LIN {X -0.082,Y -167.901,Z 1787.358,A 0.000,B 0.000,C 90.000,E1 244.409} C_DIS
LIN {X 0.085,Y -166.640,Z 1787.348,A 0.000,B 0.000,C 90.000,E1 242.615} C_DIS
LIN {X -0.008,Y -162.626,Z 1787.324,A 0.000,B 0.000,C 90.000,E1 238.280} C_DIS
LIN {X 0.050,Y -161.313,Z 1787.314,A 0.000,B 0.000,C 90.000,E1 236.501} C_DIS
LIN {X -0.040,Y -157.310,Z 1787.289,A 0.000,B 0.000,C 90.000,E1 232.110} C_DIS
LIN {X -0.106,Y -155.287,Z 1787.275,A 0.000,B 0.000,C 90.000,E1 229.461} C_DIS
LIN {X 0.041,Y -151.650,Z 1787.250,A 0.000,B 0.000,C 90.000,E1 224.919} C_DIS
LIN {X -0.022,Y -150.518,Z 1787.240,A 0.000,B 0.000,C 90.000,E1 223.137} C_DIS
LIN {X 0.001,Y -147.243,Z 1787.214,A 0.000,B 0.000,C 90.000,E1 218.588} C_DIS
LIN {X -0.034,Y -145.267,Z 1787.194,A 0.000,B 0.000,C 90.000,E1 214.945} C_DIS
LIN {X 0.000,Y -142.375,Z 1787.163,A 0.000,B 0.000,C 90.000,E1 209.411} C_DIS
LIN {X 0.049,Y -141.351,Z 1787.148,A 0.000,B 0.000,C 90.000,E1 206.616} C_DIS
LIN {X 0.033,Y -139.340,Z 1787.112,A 0.000,B 0.000,C 90.000,E1 200.120} C_DIS
LIN {X 0.082,Y -139.006,Z 1787.101,A 0.000,B 0.000,C 90.000,E1 198.236} C_DIS
LIN {X 0.039,Y -138.339,Z 1787.055,A 0.000,B 0.000,C 90.000,E1 189.849} C_DIS
LIN {X 0.061,Y -139.404,Z 1787.008,A 0.000,B 0.000,C 90.000,E1 181.432} C_DIS
LIN {X -0.025,Y -141.312,Z 1786.972,A 0.000,B 0.000,C 90.000,E1 174.951} C_DIS
LIN {X -0.068,Y -142.671,Z 1786.956,A 0.000,B 0.000,C 90.000,E1 172.186} C_DIS
LIN {X 0.054,Y -145.021,Z 1786.931,A 0.000,B 0.000,C 90.000,E1 167.521} C_DIS
LIN {X 0.011,Y -147.648,Z 1786.910,A 0.000,B 0.000,C 90.000,E1 163.866} C_DIS
LIN {X -0.053,Y -150.283,Z 1786.890,A 0.000,B 0.000,C 90.000,E1 160.242} C_DIS
LIN {X -0.040,Y -153.688,Z 1786.870,A 0.000,B 0.000,C 90.000,E1 156.613} C_DIS
LIN {X 0.015,Y -157.102,Z 1786.850,A 0.000,B 0.000,C 90.000,E1 152.999} C_DIS
LIN {X -0.047,Y -161.242,Z 1786.830,A 0.000,B 0.000,C 90.000,E1 149.459} C_DIS
LIN {X 0.038,Y -163.329,Z 1786.820,A 0.000,B 0.000,C 90.000,E1 147.661} C_DIS
LIN {X -0.091,Y -167.782,Z 1786.801,A 0.000,B 0.000,C 90.000,E1 144.196} C_DIS
LIN {X 0.061,Y -171.597,Z 1786.786,A 0.000,B 0.000,C 90.000,E1 141.537} C_DIS
LIN {X -0.009,Y -176.549,Z 1786.767,A 0.000,B 0.000,C 90.000,E1 138.119} C_DIS
LIN {X -0.017,Y -180.848,Z 1786.753,A 0.000,B 0.000,C 90.000,E1 135.567} C_DIS
LIN {X -0.033,Y -186.259,Z 1786.734,A 0.000,B 0.000,C 90.000,E1 132.204} C_DIS
LIN {X -0.096,Y -190.895,Z 1786.721,A 0.000,B 0.000,C 90.000,E1 129.725} C_DIS
LIN {X 0.095,Y -196.660,Z 1786.702,A 0.000,B 0.000,C 90.000,E1 126.377} C_DIS
LIN {X 0.013,Y -199.902,Z 1786.693,A 0.000,B 0.000,C 90.000,E1 124.771} C_DIS
LIN {X 0.045,Y -204.295,Z 1786.680,A 0.000,B 0.000,C 90.000,E1 122.339} C_DIS
LIN {X 0.080,Y -210.742,Z 1786.662,A 0.000,B 0.000,C 90.000,E1 119.077} C_DIS
LIN {X 0.011,Y -211.127,Z 1786.660,A 0.000,B 0.000,C 90.000,E1 118.871} C_DIS
LIN {X -0.018,Y -337.494,Z 1786.660,A 0.000,B 0.000,C 90.000,E1 118.871} C_DIS
LIN {X 0.027,Y -340.375,Z 1786.660,A 0.000,B 0.000,C 90.000,E1 118.821} C_DIS
LIN {X -0.117,Y -345.110,Z 1786.659,A 0.000,B 0.000,C 90.000,E1 118.615} C_DIS
LIN {X 0.042,Y -347.762,Z 1786.658,A 0.000,B 0.000,C 90.000,E1 118.359} C_DIS
LIN {X -0.138,Y -351.455,Z 1786.655,A 0.000,B 0.000,C 90.000,E1 117.897} C_DIS
LIN {X 0.053,Y -354.388,Z 1786.651,A 0.000,B 0.000,C 90.000,E1 117.257} C_DIS
LIN {X 0.173,Y -369.809,Z 1786.633,A 0.000,B 0.000,C 90.000,E1 113.951} C_DIS
LIN {X -0.041,Y -383.135,Z 1786.619,A 0.000,B 0.000,C 90.000,E1 111.354} C_DIS
LIN {X -0.205,Y -395.265,Z 1786.606,A 0.000,B 0.000,C 90.000,E1 109.087} C_DIS
LIN {X -0.242,Y -404.241,Z 1786.596,A 0.000,B 0.000,C 90.000,E1 107.402} C_DIS
LIN {X -0.047,Y -409.915,Z 1786.590,A 0.000,B 0.000,C 90.000,E1 106.260} C_DIS
LIN {X -0.008,Y -413.783,Z 1786.586,A 0.000,B 0.000,C 90.000,E1 105.426} C_DIS
LIN {X 0.107,Y -414.948,Z 1786.584,A 0.000,B 0.000,C 90.000,E1 105.134} C_DIS
LIN {X 0.061,Y -416.955,Z 1786.581,A 0.000,B 0.000,C 90.000,E1 104.592} C_DIS
LIN {X -0.085,Y -418.203,Z 1786.578,A 0.000,B 0.000,C 90.000,E1 104.064} C_DIS
LIN {X -0.218,Y -417.913,Z 1786.575,A 0.000,B 0.000,C 90.000,E1 103.536} C_DIS
LIN {X -0.102,Y -414.004,Z 1786.536,A 0.000,B 0.000,C 90.000,E1 96.543} C_DIS
LIN {X -0.164,Y -414.009,Z 1786.536,A 0.000,B 0.000,C 90.000,E1 96.543} C_DIS
LIN {X -0.056,Y -438.067,Z 1786.526,A 0.000,B 0.000,C 90.000,E1 94.702} C_DIS
LIN {X -0.081,Y -442.270,Z 1786.524,A 0.000,B 0.000,C 90.000,E1 94.302} C_DIS
LIN {X -0.189,Y -443.992,Z 1786.522,A 0.000,B 0.000,C 90.000,E1 94.069} C_DIS
LIN {X 0.112,Y -445.315,Z 1786.521,A 0.000,B 0.000,C 90.000,E1 93.784} C_DIS
LIN {X 0.030,Y -447.152,Z 1786.518,A 0.000,B 0.000,C 90.000,E1 93.269} C_DIS
LIN {X -0.018,Y -447.927,Z 1786.515,A 0.000,B 0.000,C 90.000,E1 92.751} C_DIS
LIN {X -0.078,Y -447.768,Z 1786.512,A 0.000,B 0.000,C 90.000,E1 92.236} C_DIS
LIN {X -0.117,Y -446.654,Z 1786.510,A 0.000,B 0.000,C 90.000,E1 91.718} C_DIS
LIN {X 0.078,Y -445.692,Z 1786.508,A 0.000,B 0.000,C 90.000,E1 91.432} C_DIS
LIN {X -0.171,Y -444.401,Z 1786.507,A 0.000,B 0.000,C 90.000,E1 91.203} C_DIS
LIN {X 0.183,Y -432.865,Z 1786.496,A 0.000,B 0.000,C 90.000,E1 89.312} C_DIS
LIN {X 0.182,Y -422.902,Z 1786.487,A 0.000,B 0.000,C 90.000,E1 87.707} C_DIS
LIN {X -0.204,Y -419.006,Z 1786.484,A 0.000,B 0.000,C 90.000,E1 87.135} C_DIS
LIN {X 0.152,Y -419.014,Z 1786.484,A 0.000,B 0.000,C 90.000,E1 87.078} C_DIS
LIN {X -0.079,Y -421.363,Z 1786.474,A 0.000,B 0.000,C 90.000,E1 85.298} C_DIS
LIN {X 0.158,Y -421.920,Z 1786.471,A 0.000,B 0.000,C 90.000,E1 84.723} C_DIS
LIN {X -0.020,Y -421.140,Z 1786.468,A 0.000,B 0.000,C 90.000,E1 84.204} C_DIS
LIN {X -0.192,Y -419.699,Z 1786.465,A 0.000,B 0.000,C 90.000,E1 83.685} C_DIS
LIN {X 0.047,Y -417.913,Z 1786.462,A 0.000,B 0.000,C 90.000,E1 83.109} C_DIS
LIN {X 0.133,Y -413.778,Z 1786.456,A 0.000,B 0.000,C 90.000,E1 82.008} C_DIS
LIN {X -0.185,Y -408.002,Z 1786.448,A 0.000,B 0.000,C 90.000,E1 80.679} C_DIS
LIN {X 0.058,Y -399.400,Z 1786.437,A 0.000,B 0.000,C 90.000,E1 78.701} C_DIS
LIN {X -0.110,Y -390.545,Z 1786.426,A 0.000,B 0.000,C 90.000,E1 76.756} C_DIS
LIN {X -0.075,Y -381.580,Z 1786.415,A 0.000,B 0.000,C 90.000,E1 74.755} C_DIS
LIN {X -0.040,Y -372.591,Z 1786.404,A 0.000,B 0.000,C 90.000,E1 72.725} C_DIS
LIN {X -0.081,Y -363.547,Z 1786.393,A 0.000,B 0.000,C 90.000,E1 70.678} C_DIS
LIN {X -0.076,Y -354.371,Z 1786.381,A 0.000,B 0.000,C 90.000,E1 68.592} C_DIS
LIN {X -0.155,Y -346.485,Z 1786.371,A 0.000,B 0.000,C 90.000,E1 66.794} C_DIS
LIN {X -0.098,Y -335.869,Z 1786.357,A 0.000,B 0.000,C 90.000,E1 64.332} C_DIS
LIN {X 0.061,Y -327.934,Z 1786.347,A 0.000,B 0.000,C 90.000,E1 62.436} C_DIS
LIN {X 0.073,Y -319.703,Z 1786.336,A 0.000,B 0.000,C 90.000,E1 60.539} C_DIS
LIN {X 0.090,Y -311.024,Z 1786.326,A 0.000,B 0.000,C 90.000,E1 58.614} C_DIS
LIN {X -0.149,Y -302.097,Z 1786.315,A 0.000,B 0.000,C 90.000,E1 56.707} C_DIS
LIN {X 0.034,Y -291.535,Z 1786.302,A 0.000,B 0.000,C 90.000,E1 54.356} C_DIS
LIN {X 0.051,Y -277.134,Z 1786.283,A 0.000,B 0.000,C 90.000,E1 50.964} C_DIS
LIN {X 0.048,Y -265.046,Z 1786.266,A 0.000,B 0.000,C 90.000,E1 47.838} C_DIS
LIN {X 0.015,Y -256.155,Z 1786.252,A 0.000,B 0.000,C 90.000,E1 45.364} C_DIS
LIN {X -0.042,Y -245.127,Z 1786.234,A 0.000,B 0.000,C 90.000,E1 42.123} C_DIS
LIN {X 0.016,Y -234.692,Z 1786.215,A 0.000,B 0.000,C 90.000,E1 38.785} C_DIS
LIN {X -0.115,Y -225.884,Z 1786.199,A 0.000,B 0.000,C 90.000,E1 35.804} C_DIS
LIN {X 0.031,Y -217.527,Z 1786.182,A 0.000,B 0.000,C 90.000,E1 32.704} C_DIS
LIN {X 0.027,Y -209.871,Z 1786.164,A 0.000,B 0.000,C 90.000,E1 29.589} C_DIS
LIN {X -0.029,Y -202.778,Z 1786.147,A 0.000,B 0.000,C 90.000,E1 26.437} C_DIS
LIN {X 0.022,Y -196.511,Z 1786.129,A 0.000,B 0.000,C 90.000,E1 23.206} C_DIS
LIN {X 0.044,Y -191.090,Z 1786.111,A 0.000,B 0.000,C 90.000,E1 19.939} C_DIS
LIN {X -0.077,Y -186.595,Z 1786.093,A 0.000,B 0.000,C 90.000,E1 16.677} C_DIS
LIN {X 0.071,Y -183.018,Z 1786.074,A 0.000,B 0.000,C 90.000,E1 13.300} C_DIS
LIN {X -0.098,Y -179.575,Z 1786.051,A 0.000,B 0.000,C 90.000,E1 9.151} C_DIS
LIN {X 0.079,Y -176.772,Z 1786.022,A 0.000,B 0.000,C 90.000,E1 4.012} C_DIS
LIN {X 0.045,Y -175.198,Z 1785.978,A 0.000,B 0.000,C 90.000,E1 356.102} C_DIS
LIN {X -0.039,Y -175.639,Z 1785.945,A 0.000,B 0.000,C 90.000,E1 350.151} C_DIS
LIN {X -0.007,Y -177.753,Z 1785.907,A 0.000,B 0.000,C 90.000,E1 343.323} C_DIS
LIN {X 0.010,Y -180.661,Z 1785.879,A 0.000,B 0.000,C 90.000,E1 338.230} C_DIS
LIN {X 0.016,Y -184.417,Z 1785.851,A 0.000,B 0.000,C 90.000,E1 333.179} C_DIS
LIN {X 0.042,Y -188.378,Z 1785.828,A 0.000,B 0.000,C 90.000,E1 328.997} C_DIS
LIN {X -0.070,Y -193.294,Z 1785.805,A 0.000,B 0.000,C 90.000,E1 324.895} C_DIS
LIN {X -0.058,Y -198.263,Z 1785.787,A 0.000,B 0.000,C 90.000,E1 321.618} C_DIS
LIN {X -0.021,Y -202.721,Z 1785.773,A 0.000,B 0.000,C 90.000,E1 319.175} C_DIS
LIN {X -0.077,Y -207.911,Z 1785.760,A 0.000,B 0.000,C 90.000,E1 316.782} C_DIS
LIN {X 0.113,Y -213.920,Z 1785.747,A 0.000,B 0.000,C 90.000,E1 314.352} C_DIS
LIN {X -0.080,Y -219.742,Z 1785.736,A 0.000,B 0.000,C 90.000,E1 312.447} C_DIS
LIN {X 0.064,Y -225.118,Z 1785.727,A 0.000,B 0.000,C 90.000,E1 310.862} C_DIS
LIN {X -0.093,Y -232.803,Z 1785.716,A 0.000,B 0.000,C 90.000,E1 308.991} C_DIS
LIN {X 0.081,Y -239.780,Z 1785.708,A 0.000,B 0.000,C 90.000,E1 307.443} C_DIS
LIN {X 0.052,Y -251.469,Z 1785.696,A 0.000,B 0.000,C 90.000,E1 305.231} C_DIS
LIN {X -0.046,Y -264.356,Z 1785.684,A 0.000,B 0.000,C 90.000,E1 303.086} C_DIS
LIN {X 0.077,Y -283.080,Z 1785.668,A 0.000,B 0.000,C 90.000,E1 300.256} C_DIS
LIN {X 0.015,Y -300.593,Z 1785.655,A 0.000,B 0.000,C 90.000,E1 297.897} C_DIS
LIN {X 0.114,Y -318.945,Z 1785.642,A 0.000,B 0.000,C 90.000,E1 295.591} C_DIS
LIN {X -0.054,Y -332.172,Z 1785.633,A 0.000,B 0.000,C 90.000,E1 294.027} C_DIS
LIN {X -0.015,Y -344.484,Z 1785.625,A 0.000,B 0.000,C 90.000,E1 292.514} C_DIS
LIN {X 0.041,Y -354.474,Z 1785.618,A 0.000,B 0.000,C 90.000,E1 291.280} C_DIS
LIN {X 0.098,Y -363.916,Z 1785.612,A 0.000,B 0.000,C 90.000,E1 290.066} C_DIS
LIN {X -0.153,Y -370.378,Z 1785.607,A 0.000,B 0.000,C 90.000,E1 289.214} C_DIS
LIN {X -0.001,Y -376.050,Z 1785.602,A 0.000,B 0.000,C 90.000,E1 288.308} C_DIS
LIN {X 0.213,Y -379.294,Z 1785.599,A 0.000,B 0.000,C 90.000,E1 287.692} C_DIS
LIN {X -0.033,Y -382.098,Z 1785.595,A 0.000,B 0.000,C 90.000,E1 287.149} C_DIS
LIN {X -0.007,Y -384.499,Z 1785.592,A 0.000,B 0.000,C 90.000,E1 286.567} C_DIS
LIN {X 0.150,Y -386.517,Z 1785.589,A 0.000,B 0.000,C 90.000,E1 285.969} C_DIS
LIN {X -0.061,Y -388.166,Z 1785.586,A 0.000,B 0.000,C 90.000,E1 285.426} C_DIS
LIN {X 0.113,Y -389.485,Z 1785.583,A 0.000,B 0.000,C 90.000,E1 284.828} C_DIS
LIN {X -0.180,Y -390.422,Z 1785.579,A 0.000,B 0.000,C 90.000,E1 284.300} C_DIS
LIN {X 0.008,Y -391.016,Z 1785.576,A 0.000,B 0.000,C 90.000,E1 283.703} C_DIS
LIN {X 0.110,Y -391.223,Z 1785.573,A 0.000,B 0.000,C 90.000,E1 283.119} C_DIS
LIN {X -0.164,Y -391.064,Z 1785.570,A 0.000,B 0.000,C 90.000,E1 282.591} C_DIS
LIN {X -0.054,Y -390.576,Z 1785.567,A 0.000,B 0.000,C 90.000,E1 282.007} C_DIS
LIN {X 0.056,Y -389.758,Z 1785.563,A 0.000,B 0.000,C 90.000,E1 281.422} C_DIS
LIN {X 0.162,Y -388.564,Z 1785.560,A 0.000,B 0.000,C 90.000,E1 280.838} C_DIS
LIN {X -0.120,Y -387.029,Z 1785.557,A 0.000,B 0.000,C 90.000,E1 280.310} C_DIS
LIN {X -0.052,Y -384.062,Z 1785.552,A 0.000,B 0.000,C 90.000,E1 279.443} C_DIS
LIN {X 0.051,Y -380.355,Z 1785.548,A 0.000,B 0.000,C 90.000,E1 278.568} C_DIS
LIN {X 0.055,Y -375.850,Z 1785.543,A 0.000,B 0.000,C 90.000,E1 277.701} C_DIS
LIN {X 0.024,Y -370.428,Z 1785.538,A 0.000,B 0.000,C 90.000,E1 276.834} C_DIS
LIN {X -0.037,Y -366.343,Z 1785.535,A 0.000,B 0.000,C 90.000,E1 276.258} C_DIS
LIN {X -0.119,Y -361.714,Z 1785.531,A 0.000,B 0.000,C 90.000,E1 275.682} C_DIS
LIN {X 0.129,Y -356.504,Z 1785.528,A 0.000,B 0.000,C 90.000,E1 275.049} C_DIS
LIN {X 0.065,Y -350.776,Z 1785.525,A 0.000,B 0.000,C 90.000,E1 274.473} C_DIS
LIN {X 0.104,Y -341.958,Z 1785.521,A 0.000,B 0.000,C 90.000,E1 273.669} C_DIS
LIN {X -0.056,Y -335.894,Z 1785.518,A 0.000,B 0.000,C 90.000,E1 273.212} C_DIS
LIN {X -0.008,Y -329.703,Z 1785.515,A 0.000,B 0.000,C 90.000,E1 272.751} C_DIS
LIN {X -0.105,Y -323.138,Z 1785.513,A 0.000,B 0.000,C 90.000,E1 272.350} C_DIS
LIN {X 0.043,Y -316.460,Z 1785.511,A 0.000,B 0.000,C 90.000,E1 271.949} C_DIS
LIN {X 0.136,Y -309.448,Z 1785.509,A 0.000,B 0.000,C 90.000,E1 271.604} C_DIS
LIN {X -0.089,Y -301.903,Z 1785.508,A 0.000,B 0.000,C 90.000,E1 271.375} C_DIS
LIN {X -0.015,Y -294.587,Z 1785.506,A 0.000,B 0.000,C 90.000,E1 271.146} C_DIS
LIN {X 0.115,Y -283.709,Z 1785.505,A 0.000,B 0.000,C 90.000,E1 270.859} C_DIS
LIN {X 0.130,Y -268.696,Z 1785.503,A 0.000,B 0.000,C 90.000,E1 270.573} C_DIS
LIN {X 0.081,Y -256.288,Z 1785.502,A 0.000,B 0.000,C 90.000,E1 270.401} C_DIS
LIN {X -0.121,Y -245.286,Z 1785.502,A 0.000,B 0.000,C 90.000,E1 270.344} C_DIS
LIN {X -0.078,Y -229.736,Z 1785.501,A 0.000,B 0.000,C 90.000,E1 270.286} C_DIS
LIN {X -0.083,Y -181.581,Z 1785.501,A 0.000,B 0.000,C 90.000,E1 270.286} C_DIS
LIN {X 0.088,Y -180.826,Z 1785.471,A 0.000,B 0.000,C 90.000,E1 264.837} C_DIS
LIN {X -0.012,Y -178.930,Z 1785.443,A 0.000,B 0.000,C 90.000,E1 259.803} C_DIS
LIN {X 0.026,Y -175.979,Z 1785.415,A 0.000,B 0.000,C 90.000,E1 254.700} C_DIS
LIN {X -0.028,Y -175.469,Z 1785.410,A 0.000,B 0.000,C 90.000,E1 253.866} C_DIS
LIN {X 0.028,Y -172.218,Z 1785.387,A 0.000,B 0.000,C 90.000,E1 249.571} C_DIS
LIN {X 0.006,Y -171.693,Z 1785.382,A 0.000,B 0.000,C 90.000,E1 248.720} C_DIS
LIN {X 0.081,Y -167.288,Z 1785.353,A 0.000,B 0.000,C 90.000,E1 243.512} C_DIS
LIN {X 0.014,Y -166.664,Z 1785.348,A 0.000,B 0.000,C 90.000,E1 242.666} C_DIS
LIN {X -0.070,Y -162.647,Z 1785.324,A 0.000,B 0.000,C 90.000,E1 238.329} C_DIS
LIN {X -0.008,Y -161.335,Z 1785.314,A 0.000,B 0.000,C 90.000,E1 236.548} C_DIS
LIN {X 0.035,Y -157.331,Z 1785.290,A 0.000,B 0.000,C 90.000,E1 232.110} C_DIS
LIN {X -0.032,Y -155.313,Z 1785.275,A 0.000,B 0.000,C 90.000,E1 229.461} C_DIS
LIN {X 0.007,Y -151.669,Z 1785.250,A 0.000,B 0.000,C 90.000,E1 224.960} C_DIS
LIN {X -0.053,Y -150.534,Z 1785.240,A 0.000,B 0.000,C 90.000,E1 223.176} C_DIS
LIN {X -0.020,Y -147.259,Z 1785.214,A 0.000,B 0.000,C 90.000,E1 218.624} C_DIS
LIN {X 0.037,Y -145.286,Z 1785.194,A 0.000,B 0.000,C 90.000,E1 214.945} C_DIS
LIN {X 0.071,Y -142.386,Z 1785.164,A 0.000,B 0.000,C 90.000,E1 209.411} C_DIS
LIN {X -0.007,Y -141.364,Z 1785.148,A 0.000,B 0.000,C 90.000,E1 206.668} C_DIS
LIN {X -0.028,Y -139.344,Z 1785.112,A 0.000,B 0.000,C 90.000,E1 200.174} C_DIS
LIN {X -0.023,Y -139.014,Z 1785.102,A 0.000,B 0.000,C 90.000,E1 198.308} C_DIS
LIN {X -0.028,Y -138.341,Z 1785.055,A 0.000,B 0.000,C 90.000,E1 189.905} C_DIS
LIN {X -0.008,Y -139.397,Z 1785.008,A 0.000,B 0.000,C 90.000,E1 181.489} C_DIS
LIN {X 0.045,Y -141.298,Z 1784.972,A 0.000,B 0.000,C 90.000,E1 174.951} C_DIS
LIN {X 0.003,Y -142.660,Z 1784.957,A 0.000,B 0.000,C 90.000,E1 172.186} C_DIS
LIN {X -0.047,Y -145.004,Z 1784.931,A 0.000,B 0.000,C 90.000,E1 167.589} C_DIS
LIN {X -0.057,Y -147.631,Z 1784.911,A 0.000,B 0.000,C 90.000,E1 163.921} C_DIS
LIN {X 0.020,Y -150.260,Z 1784.890,A 0.000,B 0.000,C 90.000,E1 160.242} C_DIS
LIN {X 0.033,Y -153.659,Z 1784.870,A 0.000,B 0.000,C 90.000,E1 156.613} C_DIS
LIN {X -0.050,Y -157.074,Z 1784.850,A 0.000,B 0.000,C 90.000,E1 153.050} C_DIS
LIN {X 0.029,Y -161.207,Z 1784.830,A 0.000,B 0.000,C 90.000,E1 149.459} C_DIS
LIN {X -0.023,Y -163.298,Z 1784.821,A 0.000,B 0.000,C 90.000,E1 147.709} C_DIS
LIN {X -0.013,Y -167.745,Z 1784.801,A 0.000,B 0.000,C 90.000,E1 144.196} C_DIS
LIN {X -0.101,Y -171.562,Z 1784.787,A 0.000,B 0.000,C 90.000,E1 141.618} C_DIS
LIN {X -0.060,Y -176.508,Z 1784.767,A 0.000,B 0.000,C 90.000,E1 138.162} C_DIS
LIN {X 0.065,Y -180.806,Z 1784.753,A 0.000,B 0.000,C 90.000,E1 135.567} C_DIS
LIN {X 0.051,Y -186.214,Z 1784.734,A 0.000,B 0.000,C 90.000,E1 132.204} C_DIS
LIN {X -0.011,Y -190.851,Z 1784.721,A 0.000,B 0.000,C 90.000,E1 129.725} C_DIS
LIN {X 0.023,Y -196.612,Z 1784.702,A 0.000,B 0.000,C 90.000,E1 126.423} C_DIS
LIN {X -0.064,Y -199.850,Z 1784.693,A 0.000,B 0.000,C 90.000,E1 124.818} C_DIS
LIN {X 0.132,Y -204.249,Z 1784.680,A 0.000,B 0.000,C 90.000,E1 122.339} C_DIS
LIN {X -0.043,Y -210.799,Z 1784.661,A 0.000,B 0.000,C 90.000,E1 119.077} C_DIS
LIN {X -0.001,Y -211.085,Z 1784.661,A 0.000,B 0.000,C 90.000,E1 118.899} C_DIS
LIN {X 0.125,Y -337.558,Z 1784.661,A 0.000,B 0.000,C 90.000,E1 118.871} C_DIS
LIN {X -0.126,Y -340.364,Z 1784.660,A 0.000,B 0.000,C 90.000,E1 118.871} C_DIS
LIN {X 0.030,Y -345.120,Z 1784.659,A 0.000,B 0.000,C 90.000,E1 118.615} C_DIS
LIN {X 0.189,Y -347.789,Z 1784.658,A 0.000,B 0.000,C 90.000,E1 118.359} C_DIS
LIN {X 0.024,Y -351.493,Z 1784.655,A 0.000,B 0.000,C 90.000,E1 117.897} C_DIS
LIN {X -0.097,Y -354.485,Z 1784.652,A 0.000,B 0.000,C 90.000,E1 117.308} C_DIS
LIN {X 0.015,Y -370.423,Z 1784.633,A 0.000,B 0.000,C 90.000,E1 114.003} C_DIS
LIN {X -0.053,Y -385.844,Z 1784.617,A 0.000,B 0.000,C 90.000,E1 111.099} C_DIS
LIN {X 0.221,Y -398.629,Z 1784.604,A 0.000,B 0.000,C 90.000,E1 108.779} C_DIS
LIN {X -0.048,Y -409.855,Z 1784.594,A 0.000,B 0.000,C 90.000,E1 106.858} C_DIS
LIN {X -0.059,Y -417.583,Z 1784.586,A 0.000,B 0.000,C 90.000,E1 105.481} C_DIS
LIN {X 0.189,Y -423.245,Z 1784.580,A 0.000,B 0.000,C 90.000,E1 104.356} C_DIS
LIN {X -0.174,Y -426.788,Z 1784.575,A 0.000,B 0.000,C 90.000,E1 103.592} C_DIS
LIN {X 0.159,Y -428.400,Z 1784.572,A 0.000,B 0.000,C 90.000,E1 103.008} C_DIS
LIN {X 0.084,Y -428.529,Z 1784.569,A 0.000,B 0.000,C 90.000,E1 102.479} C_DIS
LIN {X -0.001,Y -425.481,Z 1784.531,A 0.000,B 0.000,C 90.000,E1 95.625} C_DIS
LIN {X -0.063,Y -425.532,Z 1784.531,A 0.000,B 0.000,C 90.000,E1 95.625} C_DIS
LIN {X 0.160,Y -438.457,Z 1784.526,A 0.000,B 0.000,C 90.000,E1 94.645} C_DIS
LIN {X 0.132,Y -442.495,Z 1784.524,A 0.000,B 0.000,C 90.000,E1 94.245} C_DIS
LIN {X -0.029,Y -444.200,Z 1784.522,A 0.000,B 0.000,C 90.000,E1 94.012} C_DIS
LIN {X 0.222,Y -445.501,Z 1784.521,A 0.000,B 0.000,C 90.000,E1 93.726} C_DIS
LIN {X 0.143,Y -447.240,Z 1784.518,A 0.000,B 0.000,C 90.000,E1 93.212} C_DIS
LIN {X 0.095,Y -447.934,Z 1784.515,A 0.000,B 0.000,C 90.000,E1 92.694} C_DIS
LIN {X 0.037,Y -447.698,Z 1784.512,A 0.000,B 0.000,C 90.000,E1 92.178} C_DIS
LIN {X -0.003,Y -446.501,Z 1784.509,A 0.000,B 0.000,C 90.000,E1 91.661} C_DIS
LIN {X 0.192,Y -445.487,Z 1784.508,A 0.000,B 0.000,C 90.000,E1 91.375} C_DIS
LIN {X -0.058,Y -444.135,Z 1784.506,A 0.000,B 0.000,C 90.000,E1 91.146} C_DIS
LIN {X 0.012,Y -430.944,Z 1784.495,A 0.000,B 0.000,C 90.000,E1 89.026} C_DIS
LIN {X 0.149,Y -428.919,Z 1784.493,A 0.000,B 0.000,C 90.000,E1 88.682} C_DIS
LIN {X 0.086,Y -428.916,Z 1784.493,A 0.000,B 0.000,C 90.000,E1 88.682} C_DIS
LIN {X 0.132,Y -431.582,Z 1784.480,A 0.000,B 0.000,C 90.000,E1 86.331} C_DIS
LIN {X 0.006,Y -431.150,Z 1784.477,A 0.000,B 0.000,C 90.000,E1 85.812} C_DIS
LIN {X -0.149,Y -429.813,Z 1784.474,A 0.000,B 0.000,C 90.000,E1 85.298} C_DIS
LIN {X 0.154,Y -428.077,Z 1784.471,A 0.000,B 0.000,C 90.000,E1 84.723} C_DIS
LIN {X -0.113,Y -423.922,Z 1784.465,A 0.000,B 0.000,C 90.000,E1 83.685} C_DIS
LIN {X 0.131,Y -418.011,Z 1784.457,A 0.000,B 0.000,C 90.000,E1 82.299} C_DIS
LIN {X -0.010,Y -410.399,Z 1784.448,A 0.000,B 0.000,C 90.000,E1 80.679} C_DIS
LIN {X -0.116,Y -401.212,Z 1784.438,A 0.000,B 0.000,C 90.000,E1 78.757} C_DIS
LIN {X 0.138,Y -391.925,Z 1784.427,A 0.000,B 0.000,C 90.000,E1 76.756} C_DIS
LIN {X -0.175,Y -382.606,Z 1784.416,A 0.000,B 0.000,C 90.000,E1 74.810} C_DIS
LIN {X -0.113,Y -373.295,Z 1784.404,A 0.000,B 0.000,C 90.000,E1 72.779} C_DIS
LIN {X -0.136,Y -363.958,Z 1784.393,A 0.000,B 0.000,C 90.000,E1 70.732} C_DIS
LIN {X -0.118,Y -354.476,Z 1784.381,A 0.000,B 0.000,C 90.000,E1 68.646} C_DIS
LIN {X 0.155,Y -344.991,Z 1784.370,A 0.000,B 0.000,C 90.000,E1 66.485} C_DIS
LIN {X 0.163,Y -334.332,Z 1784.356,A 0.000,B 0.000,C 90.000,E1 64.024} C_DIS
LIN {X 0.096,Y -325.026,Z 1784.344,A 0.000,B 0.000,C 90.000,E1 61.847} C_DIS
LIN {X 0.133,Y -318.110,Z 1784.335,A 0.000,B 0.000,C 90.000,E1 60.255} C_DIS
LIN {X 0.125,Y -309.395,Z 1784.324,A 0.000,B 0.000,C 90.000,E1 58.329} C_DIS
LIN {X -0.139,Y -300.441,Z 1784.313,A 0.000,B 0.000,C 90.000,E1 56.421} C_DIS
LIN {X 0.161,Y -288.413,Z 1784.299,A 0.000,B 0.000,C 90.000,E1 53.703} C_DIS
LIN {X -0.026,Y -275.631,Z 1784.281,A 0.000,B 0.000,C 90.000,E1 50.678} C_DIS
LIN {X -0.067,Y -263.620,Z 1784.264,A 0.000,B 0.000,C 90.000,E1 47.553} C_DIS
LIN {X -0.138,Y -254.720,Z 1784.250,A 0.000,B 0.000,C 90.000,E1 45.081} C_DIS
LIN {X 0.129,Y -243.722,Z 1784.232,A 0.000,B 0.000,C 90.000,E1 41.757} C_DIS
LIN {X -0.041,Y -233.331,Z 1784.214,A 0.000,B 0.000,C 90.000,E1 38.463} C_DIS
LIN {X 0.100,Y -223.514,Z 1784.195,A 0.000,B 0.000,C 90.000,E1 35.025} C_DIS
LIN {X -0.122,Y -215.301,Z 1784.178,A 0.000,B 0.000,C 90.000,E1 32.005} C_DIS
LIN {X 0.076,Y -207.787,Z 1784.160,A 0.000,B 0.000,C 90.000,E1 28.821} C_DIS
LIN {X -0.027,Y -200.844,Z 1784.143,A 0.000,B 0.000,C 90.000,E1 25.668} C_DIS
LIN {X -0.104,Y -194.784,Z 1784.125,A 0.000,B 0.000,C 90.000,E1 22.461} C_DIS
LIN {X 0.055,Y -189.569,Z 1784.106,A 0.000,B 0.000,C 90.000,E1 19.141} C_DIS
LIN {X 0.017,Y -185.305,Z 1784.088,A 0.000,B 0.000,C 90.000,E1 15.843} C_DIS
LIN {X -0.090,Y -181.927,Z 1784.069,A 0.000,B 0.000,C 90.000,E1 12.535} C_DIS
LIN {X -0.052,Y -178.155,Z 1784.041,A 0.000,B 0.000,C 90.000,E1 7.466} C_DIS
LIN {X 0.029,Y -175.619,Z 1784.008,A 0.000,B 0.000,C 90.000,E1 1.489} C_DIS
LIN {X -0.083,Y -174.896,Z 1783.969,A 0.000,B 0.000,C 90.000,E1 354.432} C_DIS
LIN {X 0.043,Y -175.660,Z 1783.936,A 0.000,B 0.000,C 90.000,E1 348.409} C_DIS
LIN {X -0.041,Y -177.863,Z 1783.903,A 0.000,B 0.000,C 90.000,E1 342.472} C_DIS
LIN {X 0.049,Y -180.967,Z 1783.874,A 0.000,B 0.000,C 90.000,E1 337.358} C_DIS
LIN {X -0.102,Y -184.893,Z 1783.846,A 0.000,B 0.000,C 90.000,E1 332.359} C_DIS
LIN {X 0.020,Y -189.093,Z 1783.823,A 0.000,B 0.000,C 90.000,E1 328.152} C_DIS
LIN {X 0.014,Y -193.188,Z 1783.805,A 0.000,B 0.000,C 90.000,E1 324.848} C_DIS
LIN {X -0.014,Y -198.208,Z 1783.786,A 0.000,B 0.000,C 90.000,E1 321.582} C_DIS
LIN {X 0.030,Y -202.742,Z 1783.773,A 0.000,B 0.000,C 90.000,E1 319.138} C_DIS
LIN {X -0.018,Y -207.992,Z 1783.760,A 0.000,B 0.000,C 90.000,E1 316.743} C_DIS
LIN {X 0.029,Y -214.066,Z 1783.746,A 0.000,B 0.000,C 90.000,E1 314.352} C_DIS
LIN {X -0.002,Y -219.915,Z 1783.736,A 0.000,B 0.000,C 90.000,E1 312.405} C_DIS
LIN {X -0.020,Y -225.319,Z 1783.727,A 0.000,B 0.000,C 90.000,E1 310.862} C_DIS
LIN {X 0.025,Y -231.402,Z 1783.719,A 0.000,B 0.000,C 90.000,E1 309.322} C_DIS
LIN {X 0.031,Y -238.200,Z 1783.710,A 0.000,B 0.000,C 90.000,E1 307.810} C_DIS
LIN {X -0.027,Y -249.701,Z 1783.698,A 0.000,B 0.000,C 90.000,E1 305.598} C_DIS
LIN {X -0.014,Y -262.453,Z 1783.686,A 0.000,B 0.000,C 90.000,E1 303.420} C_DIS
LIN {X 0.057,Y -281.001,Z 1783.670,A 0.000,B 0.000,C 90.000,E1 300.590} C_DIS
LIN {X -0.060,Y -298.477,Z 1783.657,A 0.000,B 0.000,C 90.000,E1 298.231} C_DIS
LIN {X 0.023,Y -319.431,Z 1783.642,A 0.000,B 0.000,C 90.000,E1 295.591} C_DIS
LIN {X 0.014,Y -332.627,Z 1783.633,A 0.000,B 0.000,C 90.000,E1 294.003} C_DIS
LIN {X -0.093,Y -345.424,Z 1783.625,A 0.000,B 0.000,C 90.000,E1 292.461} C_DIS
LIN {X -0.026,Y -355.423,Z 1783.618,A 0.000,B 0.000,C 90.000,E1 291.227} C_DIS
LIN {X 0.168,Y -364.840,Z 1783.611,A 0.000,B 0.000,C 90.000,E1 289.993} C_DIS
LIN {X -0.076,Y -371.240,Z 1783.606,A 0.000,B 0.000,C 90.000,E1 289.141} C_DIS
LIN {X -0.016,Y -375.093,Z 1783.603,A 0.000,B 0.000,C 90.000,E1 288.544} C_DIS
LIN {X 0.074,Y -378.476,Z 1783.600,A 0.000,B 0.000,C 90.000,E1 287.946} C_DIS
LIN {X -0.057,Y -382.770,Z 1783.595,A 0.000,B 0.000,C 90.000,E1 287.094} C_DIS
LIN {X 0.085,Y -385.132,Z 1783.592,A 0.000,B 0.000,C 90.000,E1 286.496} C_DIS
LIN {X -0.129,Y -387.094,Z 1783.589,A 0.000,B 0.000,C 90.000,E1 285.953} C_DIS
LIN {X -0.069,Y -388.730,Z 1783.585,A 0.000,B 0.000,C 90.000,E1 285.371} C_DIS
LIN {X 0.109,Y -390.012,Z 1783.582,A 0.000,B 0.000,C 90.000,E1 284.773} C_DIS
LIN {X -0.179,Y -390.889,Z 1783.579,A 0.000,B 0.000,C 90.000,E1 284.245} C_DIS
LIN {X 0.014,Y -391.436,Z 1783.576,A 0.000,B 0.000,C 90.000,E1 283.647} C_DIS
LIN {X 0.119,Y -391.600,Z 1783.573,A 0.000,B 0.000,C 90.000,E1 283.063} C_DIS
LIN {X -0.152,Y -391.417,Z 1783.569,A 0.000,B 0.000,C 90.000,E1 282.535} C_DIS
LIN {X -0.039,Y -390.884,Z 1783.566,A 0.000,B 0.000,C 90.000,E1 281.951} C_DIS
LIN {X 0.073,Y -390.019,Z 1783.563,A 0.000,B 0.000,C 90.000,E1 281.366} C_DIS
LIN {X -0.200,Y -388.800,Z 1783.560,A 0.000,B 0.000,C 90.000,E1 280.838} C_DIS
LIN {X -0.097,Y -387.221,Z 1783.557,A 0.000,B 0.000,C 90.000,E1 280.254} C_DIS
LIN {X 0.037,Y -384.206,Z 1783.552,A 0.000,B 0.000,C 90.000,E1 279.378} C_DIS
LIN {X 0.079,Y -380.399,Z 1783.547,A 0.000,B 0.000,C 90.000,E1 278.511} C_DIS
LIN {X 0.083,Y -375.819,Z 1783.542,A 0.000,B 0.000,C 90.000,E1 277.644} C_DIS
LIN {X 0.053,Y -370.357,Z 1783.538,A 0.000,B 0.000,C 90.000,E1 276.777} C_DIS
LIN {X -0.032,Y -363.938,Z 1783.533,A 0.000,B 0.000,C 90.000,E1 275.910} C_DIS
LIN {X 0.156,Y -356.263,Z 1783.528,A 0.000,B 0.000,C 90.000,E1 274.992} C_DIS
LIN {X 0.136,Y -350.544,Z 1783.525,A 0.000,B 0.000,C 90.000,E1 274.416} C_DIS
LIN {X -0.028,Y -344.525,Z 1783.522,A 0.000,B 0.000,C 90.000,E1 273.898} C_DIS
LIN {X 0.063,Y -338.495,Z 1783.519,A 0.000,B 0.000,C 90.000,E1 273.383} C_DIS
LIN {X 0.025,Y -332.294,Z 1783.516,A 0.000,B 0.000,C 90.000,E1 272.922} C_DIS
LIN {X 0.135,Y -325.776,Z 1783.514,A 0.000,B 0.000,C 90.000,E1 272.465} C_DIS
LIN {X -0.138,Y -319.039,Z 1783.512,A 0.000,B 0.000,C 90.000,E1 272.121} C_DIS
LIN {X -0.135,Y -312.082,Z 1783.510,A 0.000,B 0.000,C 90.000,E1 271.776} C_DIS
LIN {X 0.137,Y -304.768,Z 1783.508,A 0.000,B 0.000,C 90.000,E1 271.432} C_DIS
LIN {X 0.122,Y -297.423,Z 1783.507,A 0.000,B 0.000,C 90.000,E1 271.203} C_DIS
LIN {X -0.106,Y -286.602,Z 1783.505,A 0.000,B 0.000,C 90.000,E1 270.974} C_DIS
LIN {X -0.105,Y -275.330,Z 1783.504,A 0.000,B 0.000,C 90.000,E1 270.745} C_DIS
LIN {X 0.058,Y -263.582,Z 1783.503,A 0.000,B 0.000,C 90.000,E1 270.516} C_DIS
LIN {X 0.030,Y -254.121,Z 1783.502,A 0.000,B 0.000,C 90.000,E1 270.401} C_DIS
LIN {X -0.073,Y -244.955,Z 1783.502,A 0.000,B 0.000,C 90.000,E1 270.344} C_DIS
LIN {X -0.032,Y -229.889,Z 1783.502,A 0.000,B 0.000,C 90.000,E1 270.286} C_DIS
LIN {X -0.046,Y -181.581,Z 1783.501,A 0.000,B 0.000,C 90.000,E1 270.286} C_DIS
LIN {X 0.085,Y -180.825,Z 1783.471,A 0.000,B 0.000,C 90.000,E1 264.837} C_DIS
LIN {X -0.016,Y -178.930,Z 1783.443,A 0.000,B 0.000,C 90.000,E1 259.803} C_DIS
LIN {X 0.022,Y -175.977,Z 1783.415,A 0.000,B 0.000,C 90.000,E1 254.700} C_DIS
LIN {X -0.033,Y -175.468,Z 1783.410,A 0.000,B 0.000,C 90.000,E1 253.866} C_DIS
LIN {X 0.024,Y -172.217,Z 1783.387,A 0.000,B 0.000,C 90.000,E1 249.571} C_DIS
LIN {X 0.001,Y -171.693,Z 1783.382,A 0.000,B 0.000,C 90.000,E1 248.720} C_DIS
LIN {X 0.077,Y -167.287,Z 1783.353,A 0.000,B 0.000,C 90.000,E1 243.512} C_DIS
LIN {X 0.010,Y -166.663,Z 1783.348,A 0.000,B 0.000,C 90.000,E1 242.666} C_DIS
LIN {X -0.073,Y -162.646,Z 1783.324,A 0.000,B 0.000,C 90.000,E1 238.329} C_DIS
LIN {X -0.011,Y -161.334,Z 1783.314,A 0.000,B 0.000,C 90.000,E1 236.548} C_DIS
LIN {X 0.031,Y -157.329,Z 1783.290,A 0.000,B 0.000,C 90.000,E1 232.110} C_DIS
LIN {X -0.036,Y -155.312,Z 1783.275,A 0.000,B 0.000,C 90.000,E1 229.461} C_DIS
LIN {X 0.003,Y -151.667,Z 1783.250,A 0.000,B 0.000,C 90.000,E1 224.960} C_DIS
LIN {X 0.047,Y -150.533,Z 1783.240,A 0.000,B 0.000,C 90.000,E1 223.137} C_DIS
LIN {X -0.023,Y -147.259,Z 1783.214,A 0.000,B 0.000,C 90.000,E1 218.624} C_DIS
LIN {X 0.034,Y -145.285,Z 1783.194,A 0.000,B 0.000,C 90.000,E1 214.945} C_DIS
LIN {X 0.068,Y -142.386,Z 1783.164,A 0.000,B 0.000,C 90.000,E1 209.411} C_DIS
LIN {X -0.010,Y -141.364,Z 1783.148,A 0.000,B 0.000,C 90.000,E1 206.668} C_DIS
LIN {X -0.033,Y -139.343,Z 1783.112,A 0.000,B 0.000,C 90.000,E1 200.174} C_DIS
LIN {X -0.027,Y -139.013,Z 1783.102,A 0.000,B 0.000,C 90.000,E1 198.308} C_DIS
LIN {X -0.032,Y -138.342,Z 1783.055,A 0.000,B 0.000,C 90.000,E1 189.905} C_DIS
LIN {X -0.012,Y -139.397,Z 1783.008,A 0.000,B 0.000,C 90.000,E1 181.489} C_DIS
LIN {X 0.042,Y -141.299,Z 1782.972,A 0.000,B 0.000,C 90.000,E1 174.951} C_DIS
LIN {X -0.001,Y -142.661,Z 1782.957,A 0.000,B 0.000,C 90.000,E1 172.186} C_DIS
LIN {X -0.051,Y -145.005,Z 1782.931,A 0.000,B 0.000,C 90.000,E1 167.589} C_DIS
LIN {X -0.062,Y -147.631,Z 1782.911,A 0.000,B 0.000,C 90.000,E1 163.921} C_DIS
LIN {X 0.016,Y -150.261,Z 1782.890,A 0.000,B 0.000,C 90.000,E1 160.242} C_DIS
LIN {X 0.031,Y -153.661,Z 1782.870,A 0.000,B 0.000,C 90.000,E1 156.613} C_DIS
LIN {X 0.087,Y -157.076,Z 1782.850,A 0.000,B 0.000,C 90.000,E1 152.999} C_DIS
LIN {X 0.026,Y -161.208,Z 1782.830,A 0.000,B 0.000,C 90.000,E1 149.459} C_DIS
LIN {X -0.027,Y -163.299,Z 1782.821,A 0.000,B 0.000,C 90.000,E1 147.709} C_DIS
LIN {X -0.016,Y -167.747,Z 1782.801,A 0.000,B 0.000,C 90.000,E1 144.196} C_DIS
LIN {X -0.105,Y -171.564,Z 1782.787,A 0.000,B 0.000,C 90.000,E1 141.618} C_DIS
LIN {X -0.064,Y -176.510,Z 1782.767,A 0.000,B 0.000,C 90.000,E1 138.162} C_DIS
LIN {X 0.061,Y -180.808,Z 1782.753,A 0.000,B 0.000,C 90.000,E1 135.567} C_DIS
LIN {X 0.046,Y -186.216,Z 1782.734,A 0.000,B 0.000,C 90.000,E1 132.204} C_DIS
LIN {X -0.015,Y -190.853,Z 1782.721,A 0.000,B 0.000,C 90.000,E1 129.725} C_DIS
LIN {X 0.019,Y -196.615,Z 1782.702,A 0.000,B 0.000,C 90.000,E1 126.423} C_DIS
LIN {X -0.069,Y -199.853,Z 1782.693,A 0.000,B 0.000,C 90.000,E1 124.818} C_DIS
LIN {X 0.128,Y -204.252,Z 1782.680,A 0.000,B 0.000,C 90.000,E1 122.339} C_DIS
LIN {X -0.048,Y -210.801,Z 1782.661,A 0.000,B 0.000,C 90.000,E1 119.077} C_DIS
LIN {X 0.049,Y -211.061,Z 1782.661,A 0.000,B 0.000,C 90.000,E1 118.899} C_DIS
LIN {X 0.034,Y -338.203,Z 1782.661,A 0.000,B 0.000,C 90.000,E1 118.899} C_DIS
LIN {X 0.169,Y -344.932,Z 1782.659,A 0.000,B 0.000,C 90.000,E1 118.615} C_DIS
LIN {X 0.181,Y -347.862,Z 1782.658,A 0.000,B 0.000,C 90.000,E1 118.359} C_DIS
LIN {X 0.000,Y -351.520,Z 1782.655,A 0.000,B 0.000,C 90.000,E1 117.897} C_DIS
LIN {X -0.089,Y -355.929,Z 1782.650,A 0.000,B 0.000,C 90.000,E1 117.001} C_DIS
LIN {X 0.084,Y -372.481,Z 1782.632,A 0.000,B 0.000,C 90.000,E1 113.695} C_DIS
LIN {X 0.090,Y -388.541,Z 1782.616,A 0.000,B 0.000,C 90.000,E1 110.791} C_DIS
LIN {X -0.071,Y -401.935,Z 1782.603,A 0.000,B 0.000,C 90.000,E1 108.544} C_DIS
LIN {X 0.129,Y -413.834,Z 1782.592,A 0.000,B 0.000,C 90.000,E1 106.567} C_DIS
LIN {X -0.081,Y -423.867,Z 1782.583,A 0.000,B 0.000,C 90.000,E1 104.954} C_DIS
LIN {X -0.169,Y -430.193,Z 1782.577,A 0.000,B 0.000,C 90.000,E1 103.883} C_DIS
LIN {X -0.056,Y -434.496,Z 1782.573,A 0.000,B 0.000,C 90.000,E1 103.063} C_DIS
LIN {X -0.095,Y -436.960,Z 1782.570,A 0.000,B 0.000,C 90.000,E1 102.535} C_DIS
LIN {X -0.120,Y -438.806,Z 1782.567,A 0.000,B 0.000,C 90.000,E1 102.007} C_DIS
LIN {X -0.137,Y -439.229,Z 1782.564,A 0.000,B 0.000,C 90.000,E1 101.478} C_DIS
LIN {X 0.092,Y -437.060,Z 1782.526,A 0.000,B 0.000,C 90.000,E1 94.759} C_DIS
LIN {X 0.028,Y -437.108,Z 1782.526,A 0.000,B 0.000,C 90.000,E1 94.759} C_DIS
LIN {X -0.121,Y -439.600,Z 1782.525,A 0.000,B 0.000,C 90.000,E1 94.588} C_DIS
LIN {X 0.069,Y -443.368,Z 1782.523,A 0.000,B 0.000,C 90.000,E1 94.131} C_DIS
LIN {X -0.176,Y -444.917,Z 1782.521,A 0.000,B 0.000,C 90.000,E1 93.898} C_DIS
LIN {X -0.009,Y -446.085,Z 1782.520,A 0.000,B 0.000,C 90.000,E1 93.612} C_DIS
LIN {X -0.060,Y -447.513,Z 1782.517,A 0.000,B 0.000,C 90.000,E1 93.094} C_DIS
LIN {X -0.128,Y -447.947,Z 1782.514,A 0.000,B 0.000,C 90.000,E1 92.579} C_DIS
LIN {X -0.185,Y -447.455,Z 1782.511,A 0.000,B 0.000,C 90.000,E1 92.064} C_DIS
LIN {X 0.222,Y -445.966,Z 1782.508,A 0.000,B 0.000,C 90.000,E1 91.489} C_DIS
LIN {X -0.029,Y -444.775,Z 1782.507,A 0.000,B 0.000,C 90.000,E1 91.260} C_DIS
LIN {X -0.037,Y -439.087,Z 1782.502,A 0.000,B 0.000,C 90.000,E1 90.344} C_DIS
LIN {X -0.100,Y -439.066,Z 1782.502,A 0.000,B 0.000,C 90.000,E1 90.344} C_DIS
LIN {X 0.062,Y -441.425,Z 1782.488,A 0.000,B 0.000,C 90.000,E1 87.822} C_DIS
LIN {X -0.033,Y -441.138,Z 1782.485,A 0.000,B 0.000,C 90.000,E1 87.306} C_DIS
LIN {X -0.103,Y -439.841,Z 1782.482,A 0.000,B 0.000,C 90.000,E1 86.788} C_DIS
LIN {X -0.198,Y -438.095,Z 1782.479,A 0.000,B 0.000,C 90.000,E1 86.274} C_DIS
LIN {X 0.078,Y -433.858,Z 1782.473,A 0.000,B 0.000,C 90.000,E1 85.179} C_DIS
LIN {X -0.002,Y -427.840,Z 1782.466,A 0.000,B 0.000,C 90.000,E1 83.856} C_DIS
LIN {X -0.118,Y -421.337,Z 1782.458,A 0.000,B 0.000,C 90.000,E1 82.527} C_DIS
LIN {X 0.217,Y -413.224,Z 1782.449,A 0.000,B 0.000,C 90.000,E1 80.849} C_DIS
LIN {X -0.207,Y -402.184,Z 1782.437,A 0.000,B 0.000,C 90.000,E1 78.701} C_DIS
LIN {X 0.066,Y -392.520,Z 1782.426,A 0.000,B 0.000,C 90.000,E1 76.700} C_DIS
LIN {X 0.131,Y -382.871,Z 1782.415,A 0.000,B 0.000,C 90.000,E1 74.700} C_DIS
LIN {X -0.175,Y -373.253,Z 1782.404,A 0.000,B 0.000,C 90.000,E1 72.725} C_DIS
LIN {X -0.081,Y -363.610,Z 1782.392,A 0.000,B 0.000,C 90.000,E1 70.659} C_DIS
LIN {X -0.142,Y -352.467,Z 1782.379,A 0.000,B 0.000,C 90.000,E1 68.284} C_DIS
LIN {X -0.081,Y -341.588,Z 1782.366,A 0.000,B 0.000,C 90.000,E1 65.845} C_DIS
LIN {X -0.146,Y -330.965,Z 1782.352,A 0.000,B 0.000,C 90.000,E1 63.384} C_DIS
LIN {X 0.065,Y -322.966,Z 1782.342,A 0.000,B 0.000,C 90.000,E1 61.463} C_DIS
LIN {X 0.066,Y -315.933,Z 1782.333,A 0.000,B 0.000,C 90.000,E1 59.871} C_DIS
LIN {X 0.014,Y -307.218,Z 1782.322,A 0.000,B 0.000,C 90.000,E1 57.946} C_DIS
LIN {X -0.125,Y -298.211,Z 1782.311,A 0.000,B 0.000,C 90.000,E1 56.008} C_DIS
LIN {X 0.033,Y -284.826,Z 1782.294,A 0.000,B 0.000,C 90.000,E1 52.970} C_DIS
LIN {X -0.070,Y -272.239,Z 1782.277,A 0.000,B 0.000,C 90.000,E1 49.908} C_DIS
LIN {X -0.018,Y -260.430,Z 1782.260,A 0.000,B 0.000,C 90.000,E1 46.743} C_DIS
LIN {X 0.039,Y -250.353,Z 1782.244,A 0.000,B 0.000,C 90.000,E1 43.866} C_DIS
LIN {X -0.154,Y -239.514,Z 1782.225,A 0.000,B 0.000,C 90.000,E1 40.620} C_DIS
LIN {X -0.061,Y -229.338,Z 1782.207,A 0.000,B 0.000,C 90.000,E1 37.237} C_DIS
LIN {X -0.083,Y -220.793,Z 1782.190,A 0.000,B 0.000,C 90.000,E1 34.199} C_DIS
LIN {X 0.001,Y -212.748,Z 1782.173,A 0.000,B 0.000,C 90.000,E1 31.082} C_DIS
LIN {X 0.035,Y -205.364,Z 1782.155,A 0.000,B 0.000,C 90.000,E1 27.924} C_DIS
LIN {X 0.056,Y -198.696,Z 1782.137,A 0.000,B 0.000,C 90.000,E1 24.719} C_DIS
LIN {X 0.029,Y -192.861,Z 1782.119,A 0.000,B 0.000,C 90.000,E1 21.482} C_DIS
LIN {X 0.076,Y -187.910,Z 1782.101,A 0.000,B 0.000,C 90.000,E1 18.181} C_DIS
LIN {X -0.052,Y -183.887,Z 1782.083,A 0.000,B 0.000,C 90.000,E1 14.898} C_DIS
LIN {X 0.094,Y -180.103,Z 1782.059,A 0.000,B 0.000,C 90.000,E1 10.658} C_DIS
LIN {X -0.044,Y -176.816,Z 1782.031,A 0.000,B 0.000,C 90.000,E1 5.625} C_DIS
LIN {X 0.001,Y -174.690,Z 1781.988,A 0.000,B 0.000,C 90.000,E1 357.822} C_DIS
LIN {X 0.027,Y -174.889,Z 1781.950,A 0.000,B 0.000,C 90.000,E1 350.971} C_DIS
LIN {X -0.025,Y -176.793,Z 1781.912,A 0.000,B 0.000,C 90.000,E1 344.157} C_DIS
LIN {X 0.069,Y -179.565,Z 1781.884,A 0.000,B 0.000,C 90.000,E1 339.028} C_DIS
LIN {X 0.046,Y -183.222,Z 1781.855,A 0.000,B 0.000,C 90.000,E1 333.973} C_DIS
LIN {X 0.028,Y -187.110,Z 1781.832,A 0.000,B 0.000,C 90.000,E1 329.793} C_DIS
LIN {X -0.066,Y -191.956,Z 1781.809,A 0.000,B 0.000,C 90.000,E1 325.674} C_DIS
LIN {X 0.068,Y -196.804,Z 1781.791,A 0.000,B 0.000,C 90.000,E1 322.351} C_DIS
LIN {X 0.081,Y -201.157,Z 1781.777,A 0.000,B 0.000,C 90.000,E1 319.908} C_DIS
LIN {X 0.004,Y -206.229,Z 1781.764,A 0.000,B 0.000,C 90.000,E1 317.514} C_DIS
LIN {X 0.016,Y -212.077,Z 1781.751,A 0.000,B 0.000,C 90.000,E1 315.121} C_DIS
LIN {X -0.053,Y -217.638,Z 1781.740,A 0.000,B 0.000,C 90.000,E1 313.176} C_DIS
LIN {X 0.047,Y -222.697,Z 1781.731,A 0.000,B 0.000,C 90.000,E1 311.595} C_DIS
LIN {X -0.088,Y -228.462,Z 1781.723,A 0.000,B 0.000,C 90.000,E1 310.092} C_DIS
LIN {X -0.017,Y -236.650,Z 1781.712,A 0.000,B 0.000,C 90.000,E1 308.177} C_DIS
LIN {X 0.051,Y -245.994,Z 1781.702,A 0.000,B 0.000,C 90.000,E1 306.297} C_DIS
LIN {X -0.004,Y -258.372,Z 1781.690,A 0.000,B 0.000,C 90.000,E1 304.119} C_DIS
LIN {X 0.107,Y -276.566,Z 1781.674,A 0.000,B 0.000,C 90.000,E1 301.258} C_DIS
LIN {X -0.119,Y -296.332,Z 1781.659,A 0.000,B 0.000,C 90.000,E1 298.565} C_DIS
LIN {X 0.013,Y -317.216,Z 1781.644,A 0.000,B 0.000,C 90.000,E1 295.899} C_DIS
LIN {X -0.168,Y -330.478,Z 1781.635,A 0.000,B 0.000,C 90.000,E1 294.335} C_DIS
LIN {X -0.166,Y -343.405,Z 1781.626,A 0.000,B 0.000,C 90.000,E1 292.770} C_DIS
LIN {X -0.103,Y -355.934,Z 1781.618,A 0.000,B 0.000,C 90.000,E1 291.227} C_DIS
LIN {X 0.097,Y -365.365,Z 1781.611,A 0.000,B 0.000,C 90.000,E1 289.993} C_DIS
LIN {X -0.145,Y -371.768,Z 1781.606,A 0.000,B 0.000,C 90.000,E1 289.141} C_DIS
LIN {X -0.081,Y -375.565,Z 1781.603,A 0.000,B 0.000,C 90.000,E1 288.544} C_DIS
LIN {X 0.011,Y -378.954,Z 1781.600,A 0.000,B 0.000,C 90.000,E1 287.946} C_DIS
LIN {X -0.116,Y -383.230,Z 1781.595,A 0.000,B 0.000,C 90.000,E1 287.094} C_DIS
LIN {X 0.029,Y -385.567,Z 1781.592,A 0.000,B 0.000,C 90.000,E1 286.496} C_DIS
LIN {X 0.190,Y -387.541,Z 1781.589,A 0.000,B 0.000,C 90.000,E1 285.898} C_DIS
LIN {X -0.120,Y -389.150,Z 1781.585,A 0.000,B 0.000,C 90.000,E1 285.371} C_DIS
LIN {X 0.060,Y -390.429,Z 1781.582,A 0.000,B 0.000,C 90.000,E1 284.773} C_DIS
LIN {X -0.226,Y -391.297,Z 1781.579,A 0.000,B 0.000,C 90.000,E1 284.245} C_DIS
LIN {X -0.031,Y -391.807,Z 1781.576,A 0.000,B 0.000,C 90.000,E1 283.647} C_DIS
LIN {X 0.077,Y -391.985,Z 1781.573,A 0.000,B 0.000,C 90.000,E1 283.063} C_DIS
LIN {X -0.192,Y -391.819,Z 1781.569,A 0.000,B 0.000,C 90.000,E1 282.535} C_DIS
LIN {X -0.076,Y -391.255,Z 1781.566,A 0.000,B 0.000,C 90.000,E1 281.951} C_DIS
LIN {X 0.039,Y -390.373,Z 1781.563,A 0.000,B 0.000,C 90.000,E1 281.366} C_DIS
LIN {X 0.150,Y -389.152,Z 1781.560,A 0.000,B 0.000,C 90.000,E1 280.782} C_DIS
LIN {X -0.128,Y -387.555,Z 1781.557,A 0.000,B 0.000,C 90.000,E1 280.254} C_DIS
LIN {X 0.009,Y -384.491,Z 1781.552,A 0.000,B 0.000,C 90.000,E1 279.378} C_DIS
LIN {X 0.055,Y -380.650,Z 1781.547,A 0.000,B 0.000,C 90.000,E1 278.511} C_DIS
LIN {X 0.062,Y -376.039,Z 1781.542,A 0.000,B 0.000,C 90.000,E1 277.644} C_DIS
LIN {X 0.031,Y -372.516,Z 1781.539,A 0.000,B 0.000,C 90.000,E1 277.068} C_DIS
LIN {X 0.024,Y -368.556,Z 1781.536,A 0.000,B 0.000,C 90.000,E1 276.486} C_DIS
LIN {X -0.049,Y -364.128,Z 1781.533,A 0.000,B 0.000,C 90.000,E1 275.910} C_DIS
LIN {X 0.142,Y -356.476,Z 1781.528,A 0.000,B 0.000,C 90.000,E1 274.992} C_DIS
LIN {X 0.066,Y -350.591,Z 1781.525,A 0.000,B 0.000,C 90.000,E1 274.416} C_DIS
LIN {X -0.065,Y -344.602,Z 1781.522,A 0.000,B 0.000,C 90.000,E1 273.898} C_DIS
LIN {X 0.042,Y -338.584,Z 1781.519,A 0.000,B 0.000,C 90.000,E1 273.383} C_DIS
LIN {X 0.096,Y -329.237,Z 1781.515,A 0.000,B 0.000,C 90.000,E1 272.694} C_DIS
LIN {X 0.061,Y -322.727,Z 1781.513,A 0.000,B 0.000,C 90.000,E1 272.293} C_DIS
LIN {X -0.052,Y -316.043,Z 1781.511,A 0.000,B 0.000,C 90.000,E1 271.949} C_DIS
LIN {X 0.095,Y -308.988,Z 1781.509,A 0.000,B 0.000,C 90.000,E1 271.604} C_DIS
LIN {X -0.088,Y -301.584,Z 1781.508,A 0.000,B 0.000,C 90.000,E1 271.375} C_DIS
LIN {X 0.097,Y -290.499,Z 1781.506,A 0.000,B 0.000,C 90.000,E1 271.031} C_DIS
LIN {X -0.027,Y -275.822,Z 1781.504,A 0.000,B 0.000,C 90.000,E1 270.745} C_DIS
LIN {X -0.121,Y -264.257,Z 1781.503,A 0.000,B 0.000,C 90.000,E1 270.573} C_DIS
LIN {X 0.119,Y -254.794,Z 1781.502,A 0.000,B 0.000,C 90.000,E1 270.401} C_DIS
LIN {X -0.079,Y -241.283,Z 1781.502,A 0.000,B 0.000,C 90.000,E1 270.344} C_DIS
LIN {X 0.024,Y -231.358,Z 1781.502,A 0.000,B 0.000,C 90.000,E1 270.286} C_DIS
LIN {X -0.002,Y -181.581,Z 1781.502,A 0.000,B 0.000,C 90.000,E1 270.286} C_DIS
LIN {X -0.032,Y -180.831,Z 1781.472,A 0.000,B 0.000,C 90.000,E1 264.894} C_DIS
LIN {X 0.048,Y -178.937,Z 1781.443,A 0.000,B 0.000,C 90.000,E1 259.803} C_DIS
LIN {X -0.084,Y -175.987,Z 1781.415,A 0.000,B 0.000,C 90.000,E1 254.755} C_DIS
LIN {X 0.030,Y -175.484,Z 1781.410,A 0.000,B 0.000,C 90.000,E1 253.866} C_DIS
LIN {X 0.087,Y -172.230,Z 1781.387,A 0.000,B 0.000,C 90.000,E1 249.571} C_DIS
LIN {X 0.064,Y -171.707,Z 1781.382,A 0.000,B 0.000,C 90.000,E1 248.720} C_DIS
LIN {X -0.011,Y -167.301,Z 1781.353,A 0.000,B 0.000,C 90.000,E1 243.563} C_DIS
LIN {X -0.005,Y -166.681,Z 1781.348,A 0.000,B 0.000,C 90.000,E1 242.692} C_DIS
LIN {X -0.014,Y -162.663,Z 1781.324,A 0.000,B 0.000,C 90.000,E1 238.329} C_DIS
LIN {X -0.040,Y -161.352,Z 1781.314,A 0.000,B 0.000,C 90.000,E1 236.580} C_DIS
LIN {X -0.006,Y -157.347,Z 1781.290,A 0.000,B 0.000,C 90.000,E1 232.145} C_DIS
LIN {X 0.022,Y -155.332,Z 1781.275,A 0.000,B 0.000,C 90.000,E1 229.461} C_DIS
LIN {X -0.047,Y -151.683,Z 1781.250,A 0.000,B 0.000,C 90.000,E1 225.000} C_DIS
LIN {X 0.001,Y -150.546,Z 1781.240,A 0.000,B 0.000,C 90.000,E1 223.176} C_DIS
LIN {X 0.034,Y -147.273,Z 1781.215,A 0.000,B 0.000,C 90.000,E1 218.624} C_DIS
LIN {X 0.006,Y -145.300,Z 1781.194,A 0.000,B 0.000,C 90.000,E1 214.978} C_DIS
LIN {X -0.002,Y -142.395,Z 1781.164,A 0.000,B 0.000,C 90.000,E1 209.461} C_DIS
LIN {X -0.018,Y -141.375,Z 1781.148,A 0.000,B 0.000,C 90.000,E1 206.693} C_DIS
LIN {X 0.023,Y -139.347,Z 1781.112,A 0.000,B 0.000,C 90.000,E1 200.174} C_DIS
LIN {X -0.036,Y -138.783,Z 1781.097,A 0.000,B 0.000,C 90.000,E1 197.402} C_DIS
LIN {X 0.023,Y -138.343,Z 1781.055,A 0.000,B 0.000,C 90.000,E1 189.905} C_DIS
LIN {X 0.043,Y -139.390,Z 1781.008,A 0.000,B 0.000,C 90.000,E1 181.489} C_DIS
LIN {X -0.043,Y -141.289,Z 1780.972,A 0.000,B 0.000,C 90.000,E1 175.008} C_DIS
LIN {X 0.056,Y -142.652,Z 1780.957,A 0.000,B 0.000,C 90.000,E1 172.186} C_DIS
LIN {X 0.005,Y -144.991,Z 1780.931,A 0.000,B 0.000,C 90.000,E1 167.589} C_DIS
LIN {X -0.005,Y -147.618,Z 1780.911,A 0.000,B 0.000,C 90.000,E1 163.921} C_DIS
LIN {X 0.073,Y -150.243,Z 1780.890,A 0.000,B 0.000,C 90.000,E1 160.242} C_DIS
LIN {X -0.053,Y -153.638,Z 1780.870,A 0.000,B 0.000,C 90.000,E1 156.666} C_DIS
LIN {X 0.006,Y -157.052,Z 1780.850,A 0.000,B 0.000,C 90.000,E1 153.050} C_DIS
LIN {X 0.003,Y -161.181,Z 1780.830,A 0.000,B 0.000,C 90.000,E1 149.488} C_DIS
LIN {X 0.034,Y -163.275,Z 1780.821,A 0.000,B 0.000,C 90.000,E1 147.709} C_DIS
LIN {X 0.045,Y -167.718,Z 1780.801,A 0.000,B 0.000,C 90.000,E1 144.196} C_DIS
LIN {X -0.043,Y -171.537,Z 1780.787,A 0.000,B 0.000,C 90.000,E1 141.618} C_DIS
LIN {X -0.001,Y -176.478,Z 1780.768,A 0.000,B 0.000,C 90.000,E1 138.162} C_DIS
LIN {X -0.001,Y -180.775,Z 1780.753,A 0.000,B 0.000,C 90.000,E1 135.607} C_DIS
LIN {X -0.013,Y -186.181,Z 1780.735,A 0.000,B 0.000,C 90.000,E1 132.243} C_DIS
LIN {X 0.051,Y -190.819,Z 1780.721,A 0.000,B 0.000,C 90.000,E1 129.725} C_DIS
LIN {X -0.030,Y -196.577,Z 1780.703,A 0.000,B 0.000,C 90.000,E1 126.457} C_DIS
LIN {X 0.055,Y -201.345,Z 1780.689,A 0.000,B 0.000,C 90.000,E1 123.992} C_DIS
LIN {X -0.017,Y -207.322,Z 1780.671,A 0.000,B 0.000,C 90.000,E1 120.797} C_DIS
LIN {X -0.066,Y -211.029,Z 1780.661,A 0.000,B 0.000,C 90.000,E1 118.949} C_DIS
LIN {X -0.149,Y -338.100,Z 1780.661,A 0.000,B 0.000,C 90.000,E1 118.949} C_DIS
LIN {X -0.185,Y -344.819,Z 1780.659,A 0.000,B 0.000,C 90.000,E1 118.693} C_DIS
LIN {X -0.009,Y -347.749,Z 1780.658,A 0.000,B 0.000,C 90.000,E1 118.409} C_DIS
LIN {X 0.118,Y -351.408,Z 1780.655,A 0.000,B 0.000,C 90.000,E1 117.897} C_DIS
LIN {X 0.029,Y -355.817,Z 1780.650,A 0.000,B 0.000,C 90.000,E1 117.001} C_DIS
LIN {X -0.122,Y -369.456,Z 1780.635,A 0.000,B 0.000,C 90.000,E1 114.335} C_DIS
LIN {X -0.062,Y -385.849,Z 1780.619,A 0.000,B 0.000,C 90.000,E1 111.408} C_DIS
LIN {X -0.100,Y -401.385,Z 1780.605,A 0.000,B 0.000,C 90.000,E1 108.852} C_DIS
LIN {X -0.074,Y -415.637,Z 1780.592,A 0.000,B 0.000,C 90.000,E1 106.622} C_DIS
LIN {X 0.154,Y -426.380,Z 1780.583,A 0.000,B 0.000,C 90.000,E1 104.954} C_DIS
LIN {X -0.142,Y -435.116,Z 1780.576,A 0.000,B 0.000,C 90.000,E1 103.647} C_DIS
LIN {X -0.204,Y -441.676,Z 1780.570,A 0.000,B 0.000,C 90.000,E1 102.591} C_DIS
LIN {X 0.022,Y -446.047,Z 1780.565,A 0.000,B 0.000,C 90.000,E1 101.771} C_DIS
LIN {X 0.049,Y -448.446,Z 1780.563,A 0.000,B 0.000,C 90.000,E1 101.243} C_DIS
LIN {X -0.155,Y -449.370,Z 1780.561,A 0.000,B 0.000,C 90.000,E1 101.007} C_DIS
LIN {X -0.191,Y -450.060,Z 1780.558,A 0.000,B 0.000,C 90.000,E1 100.489} C_DIS
LIN {X -0.198,Y -451.309,Z 1780.497,A 0.000,B 0.000,C 90.000,E1 89.542} C_DIS
LIN {X 0.218,Y -451.569,Z 1780.494,A 0.000,B 0.000,C 90.000,E1 88.969} C_DIS
LIN {X 0.183,Y -450.602,Z 1780.492,A 0.000,B 0.000,C 90.000,E1 88.453} C_DIS
LIN {X 0.163,Y -449.018,Z 1780.489,A 0.000,B 0.000,C 90.000,E1 87.936} C_DIS
LIN {X 0.124,Y -447.102,Z 1780.486,A 0.000,B 0.000,C 90.000,E1 87.421} C_DIS
LIN {X 0.035,Y -442.672,Z 1780.480,A 0.000,B 0.000,C 90.000,E1 86.388} C_DIS
LIN {X 0.080,Y -436.400,Z 1780.473,A 0.000,B 0.000,C 90.000,E1 85.065} C_DIS
LIN {X 0.164,Y -428.336,Z 1780.464,A 0.000,B 0.000,C 90.000,E1 83.457} C_DIS
LIN {X 0.196,Y -419.889,Z 1780.455,A 0.000,B 0.000,C 90.000,E1 81.837} C_DIS
LIN {X -0.197,Y -409.848,Z 1780.444,A 0.000,B 0.000,C 90.000,E1 79.982} C_DIS
LIN {X -0.148,Y -398.388,Z 1780.432,A 0.000,B 0.000,C 90.000,E1 77.757} C_DIS
LIN {X 0.100,Y -386.976,Z 1780.419,A 0.000,B 0.000,C 90.000,E1 75.463} C_DIS
LIN {X -0.106,Y -375.609,Z 1780.407,A 0.000,B 0.000,C 90.000,E1 73.196} C_DIS
LIN {X -0.084,Y -365.677,Z 1780.395,A 0.000,B 0.000,C 90.000,E1 71.148} C_DIS
LIN {X -0.042,Y -352.989,Z 1780.380,A 0.000,B 0.000,C 90.000,E1 68.465} C_DIS
LIN {X -0.109,Y -342.056,Z 1780.367,A 0.000,B 0.000,C 90.000,E1 66.049} C_DIS
LIN {X -0.020,Y -331.413,Z 1780.353,A 0.000,B 0.000,C 90.000,E1 63.563} C_DIS
LIN {X -0.084,Y -323.442,Z 1780.343,A 0.000,B 0.000,C 90.000,E1 61.691} C_DIS
LIN {X 0.054,Y -316.465,Z 1780.334,A 0.000,B 0.000,C 90.000,E1 60.078} C_DIS
LIN {X 0.173,Y -307.773,Z 1780.323,A 0.000,B 0.000,C 90.000,E1 58.122} C_DIS
LIN {X -0.121,Y -298.828,Z 1780.312,A 0.000,B 0.000,C 90.000,E1 56.215} C_DIS
LIN {X -0.093,Y -286.843,Z 1780.297,A 0.000,B 0.000,C 90.000,E1 53.543} C_DIS
LIN {X -0.027,Y -272.787,Z 1780.278,A 0.000,B 0.000,C 90.000,E1 50.114} C_DIS
LIN {X 0.057,Y -260.911,Z 1780.261,A 0.000,B 0.000,C 90.000,E1 46.944} C_DIS
LIN {X 0.098,Y -252.038,Z 1780.247,A 0.000,B 0.000,C 90.000,E1 44.433} C_DIS
LIN {X 0.114,Y -241.065,Z 1780.229,A 0.000,B 0.000,C 90.000,E1 41.148} C_DIS
LIN {X 0.054,Y -230.794,Z 1780.210,A 0.000,B 0.000,C 90.000,E1 37.810} C_DIS
LIN {X -0.003,Y -221.062,Z 1780.191,A 0.000,B 0.000,C 90.000,E1 34.405} C_DIS
LIN {X -0.099,Y -212.982,Z 1780.174,A 0.000,B 0.000,C 90.000,E1 31.337} C_DIS
LIN {X 0.039,Y -205.534,Z 1780.156,A 0.000,B 0.000,C 90.000,E1 28.153} C_DIS
LIN {X 0.056,Y -198.823,Z 1780.139,A 0.000,B 0.000,C 90.000,E1 24.951} C_DIS
LIN {X 0.024,Y -192.926,Z 1780.121,A 0.000,B 0.000,C 90.000,E1 21.716} C_DIS
LIN {X 0.068,Y -187.904,Z 1780.102,A 0.000,B 0.000,C 90.000,E1 18.417} C_DIS
LIN {X -0.062,Y -183.840,Z 1780.084,A 0.000,B 0.000,C 90.000,E1 15.134} C_DIS
LIN {X 0.083,Y -179.971,Z 1780.061,A 0.000,B 0.000,C 90.000,E1 10.894} C_DIS
LIN {X -0.037,Y -176.621,Z 1780.032,A 0.000,B 0.000,C 90.000,E1 5.853} C_DIS
LIN {X -0.019,Y -174.474,Z 1779.993,A 0.000,B 0.000,C 90.000,E1 358.682} C_DIS
LIN {X -0.025,Y -174.482,Z 1779.955,A 0.000,B 0.000,C 90.000,E1 351.837} C_DIS
LIN {X -0.058,Y -176.506,Z 1779.912,A 0.000,B 0.000,C 90.000,E1 344.157} C_DIS
LIN {X 0.025,Y -179.290,Z 1779.884,A 0.000,B 0.000,C 90.000,E1 339.028} C_DIS
LIN {X -0.010,Y -182.964,Z 1779.855,A 0.000,B 0.000,C 90.000,E1 333.973} C_DIS
LIN {X -0.036,Y -186.911,Z 1779.832,A 0.000,B 0.000,C 90.000,E1 329.793} C_DIS
LIN {X -0.029,Y -191.829,Z 1779.809,A 0.000,B 0.000,C 90.000,E1 325.642} C_DIS
LIN {X -0.009,Y -196.770,Z 1779.791,A 0.000,B 0.000,C 90.000,E1 322.351} C_DIS
LIN {X 0.002,Y -201.169,Z 1779.777,A 0.000,B 0.000,C 90.000,E1 319.908} C_DIS
LIN {X 0.075,Y -206.302,Z 1779.764,A 0.000,B 0.000,C 90.000,E1 317.472} C_DIS
LIN {X 0.083,Y -212.213,Z 1779.751,A 0.000,B 0.000,C 90.000,E1 315.081} C_DIS
LIN {X 0.014,Y -217.793,Z 1779.740,A 0.000,B 0.000,C 90.000,E1 313.137} C_DIS
LIN {X -0.035,Y -222.878,Z 1779.731,A 0.000,B 0.000,C 90.000,E1 311.595} C_DIS
LIN {X 0.005,Y -228.674,Z 1779.723,A 0.000,B 0.000,C 90.000,E1 310.048} C_DIS
LIN {X -0.097,Y -236.885,Z 1779.712,A 0.000,B 0.000,C 90.000,E1 308.177} C_DIS
LIN {X -0.041,Y -248.237,Z 1779.700,A 0.000,B 0.000,C 90.000,E1 305.931} C_DIS
LIN {X 0.155,Y -260.869,Z 1779.688,A 0.000,B 0.000,C 90.000,E1 303.706} C_DIS
LIN {X -0.039,Y -279.339,Z 1779.672,A 0.000,B 0.000,C 90.000,E1 300.924} C_DIS
LIN {X -0.050,Y -296.746,Z 1779.658,A 0.000,B 0.000,C 90.000,E1 298.537} C_DIS
LIN {X -0.005,Y -317.624,Z 1779.644,A 0.000,B 0.000,C 90.000,E1 295.899} C_DIS
LIN {X -0.173,Y -330.824,Z 1779.635,A 0.000,B 0.000,C 90.000,E1 294.335} C_DIS
LIN {X -0.161,Y -341.247,Z 1779.628,A 0.000,B 0.000,C 90.000,E1 293.078} C_DIS
LIN {X -0.123,Y -353.844,Z 1779.620,A 0.000,B 0.000,C 90.000,E1 291.535} C_DIS
LIN {X 0.050,Y -363.467,Z 1779.613,A 0.000,B 0.000,C 90.000,E1 290.301} C_DIS
LIN {X 0.134,Y -370.146,Z 1779.608,A 0.000,B 0.000,C 90.000,E1 289.396} C_DIS
LIN {X -0.163,Y -374.141,Z 1779.605,A 0.000,B 0.000,C 90.000,E1 288.852} C_DIS
LIN {X 0.038,Y -377.722,Z 1779.601,A 0.000,B 0.000,C 90.000,E1 288.236} C_DIS
LIN {X 0.145,Y -380.882,Z 1779.598,A 0.000,B 0.000,C 90.000,E1 287.638} C_DIS
LIN {X -0.091,Y -383.632,Z 1779.595,A 0.000,B 0.000,C 90.000,E1 287.094} C_DIS
LIN {X 0.056,Y -385.956,Z 1779.592,A 0.000,B 0.000,C 90.000,E1 286.496} C_DIS
LIN {X 0.220,Y -387.964,Z 1779.589,A 0.000,B 0.000,C 90.000,E1 285.898} C_DIS
LIN {X -0.087,Y -389.523,Z 1779.585,A 0.000,B 0.000,C 90.000,E1 285.371} C_DIS
LIN {X 0.095,Y -390.790,Z 1779.582,A 0.000,B 0.000,C 90.000,E1 284.773} C_DIS
LIN {X -0.189,Y -391.675,Z 1779.579,A 0.000,B 0.000,C 90.000,E1 284.245} C_DIS
LIN {X 0.009,Y -392.175,Z 1779.576,A 0.000,B 0.000,C 90.000,E1 283.647} C_DIS
LIN {X 0.119,Y -392.322,Z 1779.573,A 0.000,B 0.000,C 90.000,E1 283.063} C_DIS
LIN {X -0.148,Y -392.195,Z 1779.570,A 0.000,B 0.000,C 90.000,E1 282.535} C_DIS
LIN {X -0.030,Y -391.629,Z 1779.566,A 0.000,B 0.000,C 90.000,E1 281.951} C_DIS
LIN {X 0.087,Y -390.744,Z 1779.563,A 0.000,B 0.000,C 90.000,E1 281.366} C_DIS
LIN {X -0.183,Y -389.502,Z 1779.560,A 0.000,B 0.000,C 90.000,E1 280.838} C_DIS
LIN {X -0.075,Y -387.893,Z 1779.557,A 0.000,B 0.000,C 90.000,E1 280.254} C_DIS
LIN {X 0.065,Y -384.794,Z 1779.552,A 0.000,B 0.000,C 90.000,E1 279.378} C_DIS
LIN {X 0.112,Y -380.936,Z 1779.547,A 0.000,B 0.000,C 90.000,E1 278.511} C_DIS
LIN {X 0.122,Y -376.314,Z 1779.543,A 0.000,B 0.000,C 90.000,E1 277.644} C_DIS
LIN {X 0.091,Y -372.789,Z 1779.539,A 0.000,B 0.000,C 90.000,E1 277.068} C_DIS
LIN {X 0.035,Y -366.706,Z 1779.534,A 0.000,B 0.000,C 90.000,E1 276.201} C_DIS
LIN {X -0.046,Y -362.019,Z 1779.531,A 0.000,B 0.000,C 90.000,E1 275.625} C_DIS
LIN {X -0.149,Y -356.740,Z 1779.528,A 0.000,B 0.000,C 90.000,E1 275.049} C_DIS
LIN {X -0.170,Y -350.919,Z 1779.525,A 0.000,B 0.000,C 90.000,E1 274.473} C_DIS
LIN {X -0.022,Y -342.105,Z 1779.520,A 0.000,B 0.000,C 90.000,E1 273.669} C_DIS
LIN {X -0.150,Y -336.007,Z 1779.518,A 0.000,B 0.000,C 90.000,E1 273.212} C_DIS
LIN {X -0.067,Y -329.702,Z 1779.515,A 0.000,B 0.000,C 90.000,E1 272.751} C_DIS
LIN {X -0.103,Y -323.188,Z 1779.513,A 0.000,B 0.000,C 90.000,E1 272.350} C_DIS
LIN {X 0.095,Y -316.529,Z 1779.511,A 0.000,B 0.000,C 90.000,E1 271.949} C_DIS
LIN {X -0.085,Y -309.415,Z 1779.509,A 0.000,B 0.000,C 90.000,E1 271.661} C_DIS
LIN {X 0.023,Y -302.051,Z 1779.508,A 0.000,B 0.000,C 90.000,E1 271.375} C_DIS
LIN {X -0.104,Y -291.008,Z 1779.506,A 0.000,B 0.000,C 90.000,E1 271.088} C_DIS
LIN {X 0.121,Y -280.010,Z 1779.505,A 0.000,B 0.000,C 90.000,E1 270.802} C_DIS
LIN {X -0.042,Y -268.609,Z 1779.503,A 0.000,B 0.000,C 90.000,E1 270.630} C_DIS
LIN {X -0.088,Y -259.929,Z 1779.503,A 0.000,B 0.000,C 90.000,E1 270.516} C_DIS
LIN {X 0.074,Y -245.319,Z 1779.502,A 0.000,B 0.000,C 90.000,E1 270.344} C_DIS
LIN {X 0.084,Y -232.581,Z 1779.502,A 0.000,B 0.000,C 90.000,E1 270.286} C_DIS
LIN {X 0.046,Y -181.581,Z 1779.502,A 0.000,B 0.000,C 90.000,E1 270.286} C_DIS
LIN {X 0.018,Y -180.836,Z 1779.472,A 0.000,B 0.000,C 90.000,E1 264.894} C_DIS
LIN {X 0.097,Y -178.943,Z 1779.443,A 0.000,B 0.000,C 90.000,E1 259.803} C_DIS
LIN {X -0.036,Y -175.994,Z 1779.415,A 0.000,B 0.000,C 90.000,E1 254.755} C_DIS
LIN {X -0.090,Y -175.497,Z 1779.411,A 0.000,B 0.000,C 90.000,E1 253.921} C_DIS
LIN {X -0.027,Y -172.239,Z 1779.387,A 0.000,B 0.000,C 90.000,E1 249.625} C_DIS
LIN {X -0.048,Y -171.718,Z 1779.382,A 0.000,B 0.000,C 90.000,E1 248.773} C_DIS
LIN {X -0.038,Y -167.312,Z 1779.353,A 0.000,B 0.000,C 90.000,E1 243.589} C_DIS
LIN {X 0.042,Y -166.694,Z 1779.348,A 0.000,B 0.000,C 90.000,E1 242.692} C_DIS
LIN {X 0.033,Y -162.675,Z 1779.324,A 0.000,B 0.000,C 90.000,E1 238.329} C_DIS
LIN {X 0.006,Y -161.366,Z 1779.314,A 0.000,B 0.000,C 90.000,E1 236.580} C_DIS
LIN {X -0.085,Y -157.360,Z 1779.290,A 0.000,B 0.000,C 90.000,E1 232.190} C_DIS
LIN {X 0.068,Y -155.349,Z 1779.275,A 0.000,B 0.000,C 90.000,E1 229.461} C_DIS
LIN {X -0.003,Y -151.694,Z 1779.250,A 0.000,B 0.000,C 90.000,E1 225.000} C_DIS
LIN {X 0.046,Y -150.556,Z 1779.240,A 0.000,B 0.000,C 90.000,E1 223.176} C_DIS
LIN {X -0.038,Y -147.283,Z 1779.215,A 0.000,B 0.000,C 90.000,E1 218.669} C_DIS
LIN {X -0.070,Y -145.312,Z 1779.194,A 0.000,B 0.000,C 90.000,E1 215.025} C_DIS
LIN {X 0.041,Y -142.400,Z 1779.164,A 0.000,B 0.000,C 90.000,E1 209.461} C_DIS
LIN {X 0.024,Y -141.383,Z 1779.148,A 0.000,B 0.000,C 90.000,E1 206.693} C_DIS
LIN {X 0.016,Y -139.349,Z 1779.112,A 0.000,B 0.000,C 90.000,E1 200.194} C_DIS
LIN {X 0.007,Y -138.787,Z 1779.097,A 0.000,B 0.000,C 90.000,E1 197.402} C_DIS
LIN {X 0.065,Y -138.344,Z 1779.055,A 0.000,B 0.000,C 90.000,E1 189.905} C_DIS
LIN {X -0.054,Y -139.385,Z 1779.008,A 0.000,B 0.000,C 90.000,E1 181.547} C_DIS
LIN {X -0.001,Y -141.281,Z 1778.972,A 0.000,B 0.000,C 90.000,E1 175.008} C_DIS
LIN {X -0.043,Y -142.645,Z 1778.957,A 0.000,B 0.000,C 90.000,E1 172.243} C_DIS
LIN {X 0.049,Y -144.980,Z 1778.931,A 0.000,B 0.000,C 90.000,E1 167.589} C_DIS
LIN {X 0.040,Y -147.607,Z 1778.911,A 0.000,B 0.000,C 90.000,E1 163.921} C_DIS
LIN {X -0.023,Y -150.229,Z 1778.891,A 0.000,B 0.000,C 90.000,E1 160.296} C_DIS
LIN {X -0.007,Y -153.620,Z 1778.870,A 0.000,B 0.000,C 90.000,E1 156.666} C_DIS
LIN {X -0.020,Y -157.036,Z 1778.850,A 0.000,B 0.000,C 90.000,E1 153.076} C_DIS
LIN {X -0.089,Y -161.161,Z 1778.831,A 0.000,B 0.000,C 90.000,E1 149.537} C_DIS
LIN {X -0.006,Y -163.256,Z 1778.821,A 0.000,B 0.000,C 90.000,E1 147.740} C_DIS
LIN {X 0.092,Y -167.695,Z 1778.801,A 0.000,B 0.000,C 90.000,E1 144.196} C_DIS
LIN {X 0.006,Y -171.516,Z 1778.787,A 0.000,B 0.000,C 90.000,E1 141.618} C_DIS
LIN {X 0.049,Y -176.452,Z 1778.768,A 0.000,B 0.000,C 90.000,E1 138.162} C_DIS
LIN {X -0.081,Y -180.749,Z 1778.753,A 0.000,B 0.000,C 90.000,E1 135.648} C_DIS
LIN {X 0.037,Y -186.154,Z 1778.735,A 0.000,B 0.000,C 90.000,E1 132.243} C_DIS
LIN {X -0.044,Y -190.791,Z 1778.721,A 0.000,B 0.000,C 90.000,E1 129.769} C_DIS
LIN {X 0.022,Y -196.548,Z 1778.703,A 0.000,B 0.000,C 90.000,E1 126.457} C_DIS
LIN {X -0.059,Y -201.320,Z 1778.689,A 0.000,B 0.000,C 90.000,E1 124.040} C_DIS
LIN {X 0.036,Y -207.292,Z 1778.671,A 0.000,B 0.000,C 90.000,E1 120.797} C_DIS
LIN {X 0.016,Y -210.990,Z 1778.661,A 0.000,B 0.000,C 90.000,E1 118.949} C_DIS
LIN {X -0.019,Y -337.861,Z 1778.661,A 0.000,B 0.000,C 90.000,E1 118.949} C_DIS
LIN {X -0.106,Y -338.959,Z 1778.661,A 0.000,B 0.000,C 90.000,E1 118.949} C_DIS
LIN {X -0.096,Y -344.780,Z 1778.659,A 0.000,B 0.000,C 90.000,E1 118.693} C_DIS
LIN {X -0.085,Y -347.684,Z 1778.658,A 0.000,B 0.000,C 90.000,E1 118.437} C_DIS
LIN {X 0.187,Y -351.345,Z 1778.655,A 0.000,B 0.000,C 90.000,E1 117.897} C_DIS
LIN {X -0.187,Y -357.184,Z 1778.648,A 0.000,B 0.000,C 90.000,E1 116.744} C_DIS
LIN {X 0.036,Y -370.991,Z 1778.634,A 0.000,B 0.000,C 90.000,E1 114.027} C_DIS
LIN {X -0.062,Y -389.714,Z 1778.616,A 0.000,B 0.000,C 90.000,E1 110.844} C_DIS
LIN {X -0.125,Y -405.936,Z 1778.602,A 0.000,B 0.000,C 90.000,E1 108.308} C_DIS
LIN {X 0.012,Y -420.863,Z 1778.589,A 0.000,B 0.000,C 90.000,E1 106.079} C_DIS
LIN {X 0.091,Y -434.067,Z 1778.579,A 0.000,B 0.000,C 90.000,E1 104.175} C_DIS
LIN {X -0.199,Y -443.322,Z 1778.571,A 0.000,B 0.000,C 90.000,E1 102.883} C_DIS
LIN {X -0.165,Y -450.366,Z 1778.566,A 0.000,B 0.000,C 90.000,E1 101.827} C_DIS
LIN {X 0.136,Y -455.190,Z 1778.561,A 0.000,B 0.000,C 90.000,E1 101.007} C_DIS
LIN {X 0.131,Y -457.995,Z 1778.558,A 0.000,B 0.000,C 90.000,E1 100.489} C_DIS
LIN {X 0.227,Y -460.186,Z 1778.556,A 0.000,B 0.000,C 90.000,E1 99.962} C_DIS
LIN {X -0.194,Y -461.003,Z 1778.553,A 0.000,B 0.000,C 90.000,E1 99.500} C_DIS
LIN {X 0.060,Y -461.856,Z 1778.504,A 0.000,B 0.000,C 90.000,E1 90.745} C_DIS
LIN {X 0.087,Y -461.608,Z 1778.501,A 0.000,B 0.000,C 90.000,E1 90.229} C_DIS
LIN {X 0.115,Y -460.308,Z 1778.499,A 0.000,B 0.000,C 90.000,E1 89.714} C_DIS
LIN {X 0.141,Y -458.539,Z 1778.496,A 0.000,B 0.000,C 90.000,E1 89.198} C_DIS
LIN {X -0.067,Y -455.405,Z 1778.491,A 0.000,B 0.000,C 90.000,E1 88.453} C_DIS
LIN {X -0.071,Y -450.675,Z 1778.486,A 0.000,B 0.000,C 90.000,E1 87.421} C_DIS
LIN {X 0.063,Y -444.195,Z 1778.478,A 0.000,B 0.000,C 90.000,E1 86.102} C_DIS
LIN {X 0.125,Y -437.249,Z 1778.471,A 0.000,B 0.000,C 90.000,E1 84.780} C_DIS
LIN {X -0.161,Y -428.616,Z 1778.462,A 0.000,B 0.000,C 90.000,E1 83.223} C_DIS
LIN {X -0.022,Y -418.259,Z 1778.452,A 0.000,B 0.000,C 90.000,E1 81.319} C_DIS
LIN {X 0.021,Y -407.805,Z 1778.441,A 0.000,B 0.000,C 90.000,E1 79.398} C_DIS
LIN {X 0.015,Y -395.982,Z 1778.429,A 0.000,B 0.000,C 90.000,E1 77.173} C_DIS
LIN {X -0.181,Y -384.222,Z 1778.416,A 0.000,B 0.000,C 90.000,E1 74.936} C_DIS
LIN {X 0.015,Y -372.514,Z 1778.403,A 0.000,B 0.000,C 90.000,E1 72.598} C_DIS
LIN {X 0.044,Y -361.048,Z 1778.390,A 0.000,B 0.000,C 90.000,E1 70.242} C_DIS
LIN {X 0.078,Y -348.479,Z 1778.375,A 0.000,B 0.000,C 90.000,E1 67.539} C_DIS
LIN {X 0.028,Y -336.262,Z 1778.360,A 0.000,B 0.000,C 90.000,E1 64.793} C_DIS
LIN {X 0.009,Y -327.004,Z 1778.348,A 0.000,B 0.000,C 90.000,E1 62.615} C_DIS
LIN {X -0.078,Y -320.281,Z 1778.339,A 0.000,B 0.000,C 90.000,E1 61.051} C_DIS
LIN {X -0.041,Y -311.763,Z 1778.328,A 0.000,B 0.000,C 90.000,E1 59.125} C_DIS
LIN {X -0.001,Y -302.947,Z 1778.318,A 0.000,B 0.000,C 90.000,E1 57.168} C_DIS
LIN {X 0.033,Y -293.909,Z 1778.307,A 0.000,B 0.000,C 90.000,E1 55.182} C_DIS
LIN {X -0.041,Y -279.336,Z 1778.288,A 0.000,B 0.000,C 90.000,E1 51.823} C_DIS
LIN {X -0.025,Y -268.369,Z 1778.272,A 0.000,B 0.000,C 90.000,E1 49.057} C_DIS
LIN {X -0.079,Y -256.746,Z 1778.255,A 0.000,B 0.000,C 90.000,E1 45.891} C_DIS
LIN {X 0.061,Y -245.487,Z 1778.237,A 0.000,B 0.000,C 90.000,E1 42.609} C_DIS
LIN {X 0.096,Y -234.869,Z 1778.218,A 0.000,B 0.000,C 90.000,E1 39.277} C_DIS
LIN {X -0.039,Y -225.922,Z 1778.202,A 0.000,B 0.000,C 90.000,E1 36.297} C_DIS
LIN {X 0.043,Y -217.542,Z 1778.185,A 0.000,B 0.000,C 90.000,E1 33.214} C_DIS
LIN {X -0.074,Y -209.684,Z 1778.167,A 0.000,B 0.000,C 90.000,E1 30.129} C_DIS
LIN {X -0.035,Y -202.540,Z 1778.150,A 0.000,B 0.000,C 90.000,E1 26.950} C_DIS
LIN {X 0.092,Y -196.144,Z 1778.132,A 0.000,B 0.000,C 90.000,E1 23.695} C_DIS
LIN {X -0.077,Y -190.592,Z 1778.114,A 0.000,B 0.000,C 90.000,E1 20.482} C_DIS
LIN {X 0.023,Y -185.899,Z 1778.095,A 0.000,B 0.000,C 90.000,E1 17.149} C_DIS
LIN {X -0.028,Y -182.197,Z 1778.077,A 0.000,B 0.000,C 90.000,E1 13.828} C_DIS
LIN {X -0.011,Y -178.654,Z 1778.053,A 0.000,B 0.000,C 90.000,E1 9.613} C_DIS
LIN {X -0.045,Y -175.703,Z 1778.025,A 0.000,B 0.000,C 90.000,E1 4.531} C_DIS
LIN {X 0.014,Y -173.971,Z 1777.978,A 0.000,B 0.000,C 90.000,E1 356.102} C_DIS
LIN {X 0.051,Y -174.456,Z 1777.945,A 0.000,B 0.000,C 90.000,E1 350.095} C_DIS
LIN {X 0.022,Y -176.601,Z 1777.907,A 0.000,B 0.000,C 90.000,E1 343.268} C_DIS
LIN {X 0.059,Y -179.594,Z 1777.879,A 0.000,B 0.000,C 90.000,E1 338.156} C_DIS
LIN {X -0.049,Y -183.438,Z 1777.851,A 0.000,B 0.000,C 90.000,E1 333.127} C_DIS
LIN {X -0.061,Y -187.632,Z 1777.827,A 0.000,B 0.000,C 90.000,E1 328.948} C_DIS
LIN {X 0.059,Y -191.718,Z 1777.809,A 0.000,B 0.000,C 90.000,E1 325.595} C_DIS
LIN {X -0.083,Y -196.734,Z 1777.791,A 0.000,B 0.000,C 90.000,E1 322.351} C_DIS
LIN {X -0.054,Y -202.822,Z 1777.773,A 0.000,B 0.000,C 90.000,E1 319.094} C_DIS
LIN {X -0.084,Y -209.246,Z 1777.757,A 0.000,B 0.000,C 90.000,E1 316.296} C_DIS
LIN {X 0.144,Y -215.618,Z 1777.744,A 0.000,B 0.000,C 90.000,E1 313.866} C_DIS
LIN {X -0.091,Y -220.422,Z 1777.735,A 0.000,B 0.000,C 90.000,E1 312.366} C_DIS
LIN {X 0.062,Y -225.873,Z 1777.727,A 0.000,B 0.000,C 90.000,E1 310.782} C_DIS
LIN {X -0.032,Y -232.062,Z 1777.718,A 0.000,B 0.000,C 90.000,E1 309.277} C_DIS
LIN {X 0.133,Y -238.910,Z 1777.710,A 0.000,B 0.000,C 90.000,E1 307.729} C_DIS
LIN {X 0.091,Y -250.512,Z 1777.697,A 0.000,B 0.000,C 90.000,E1 305.518} C_DIS
LIN {X 0.015,Y -265.647,Z 1777.683,A 0.000,B 0.000,C 90.000,E1 303.007} C_DIS
LIN {X 0.031,Y -284.541,Z 1777.668,A 0.000,B 0.000,C 90.000,E1 300.207} C_DIS
LIN {X 0.000,Y -299.670,Z 1777.657,A 0.000,B 0.000,C 90.000,E1 298.180} C_DIS
LIN {X -0.069,Y -318.075,Z 1777.644,A 0.000,B 0.000,C 90.000,E1 295.899} C_DIS
LIN {X 0.067,Y -331.260,Z 1777.635,A 0.000,B 0.000,C 90.000,E1 294.283} C_DIS
LIN {X 0.093,Y -343.823,Z 1777.627,A 0.000,B 0.000,C 90.000,E1 292.770} C_DIS
LIN {X 0.144,Y -355.963,Z 1777.618,A 0.000,B 0.000,C 90.000,E1 291.280} C_DIS
LIN {X -0.178,Y -363.189,Z 1777.613,A 0.000,B 0.000,C 90.000,E1 290.429} C_DIS
LIN {X 0.025,Y -369.917,Z 1777.608,A 0.000,B 0.000,C 90.000,E1 289.504} C_DIS
LIN {X 0.076,Y -373.956,Z 1777.605,A 0.000,B 0.000,C 90.000,E1 288.906} C_DIS
LIN {X -0.200,Y -377.602,Z 1777.602,A 0.000,B 0.000,C 90.000,E1 288.362} C_DIS
LIN {X -0.095,Y -380.815,Z 1777.599,A 0.000,B 0.000,C 90.000,E1 287.764} C_DIS
LIN {X 0.035,Y -383.624,Z 1777.595,A 0.000,B 0.000,C 90.000,E1 287.166} C_DIS
LIN {X -0.185,Y -386.003,Z 1777.592,A 0.000,B 0.000,C 90.000,E1 286.622} C_DIS
LIN {X -0.020,Y -388.033,Z 1777.589,A 0.000,B 0.000,C 90.000,E1 286.024} C_DIS
LIN {X 0.152,Y -389.685,Z 1777.586,A 0.000,B 0.000,C 90.000,E1 285.426} C_DIS
LIN {X -0.143,Y -390.984,Z 1777.583,A 0.000,B 0.000,C 90.000,E1 284.898} C_DIS
LIN {X 0.051,Y -391.924,Z 1777.579,A 0.000,B 0.000,C 90.000,E1 284.300} C_DIS
LIN {X -0.224,Y -392.495,Z 1777.576,A 0.000,B 0.000,C 90.000,E1 283.772} C_DIS
LIN {X -0.022,Y -392.727,Z 1777.573,A 0.000,B 0.000,C 90.000,E1 283.175} C_DIS
LIN {X 0.095,Y -392.608,Z 1777.570,A 0.000,B 0.000,C 90.000,E1 282.591} C_DIS
LIN {X -0.170,Y -392.111,Z 1777.567,A 0.000,B 0.000,C 90.000,E1 282.063} C_DIS
LIN {X -0.051,Y -391.263,Z 1777.564,A 0.000,B 0.000,C 90.000,E1 281.478} C_DIS
LIN {X 0.064,Y -390.067,Z 1777.561,A 0.000,B 0.000,C 90.000,E1 280.894} C_DIS
LIN {X 0.172,Y -388.479,Z 1777.557,A 0.000,B 0.000,C 90.000,E1 280.310} C_DIS
LIN {X -0.129,Y -385.428,Z 1777.553,A 0.000,B 0.000,C 90.000,E1 279.500} C_DIS
LIN {X -0.013,Y -381.612,Z 1777.548,A 0.000,B 0.000,C 90.000,E1 278.624} C_DIS
LIN {X 0.002,Y -377.016,Z 1777.543,A 0.000,B 0.000,C 90.000,E1 277.757} C_DIS
LIN {X -0.018,Y -371.692,Z 1777.538,A 0.000,B 0.000,C 90.000,E1 276.891} C_DIS
LIN {X -0.073,Y -367.644,Z 1777.535,A 0.000,B 0.000,C 90.000,E1 276.315} C_DIS
LIN {X -0.147,Y -363.050,Z 1777.532,A 0.000,B 0.000,C 90.000,E1 275.739} C_DIS
LIN {X 0.111,Y -357.805,Z 1777.528,A 0.000,B 0.000,C 90.000,E1 275.106} C_DIS
LIN {X 0.058,Y -352.051,Z 1777.525,A 0.000,B 0.000,C 90.000,E1 274.531} C_DIS
LIN {X -0.060,Y -346.171,Z 1777.522,A 0.000,B 0.000,C 90.000,E1 274.012} C_DIS
LIN {X 0.016,Y -340.134,Z 1777.519,A 0.000,B 0.000,C 90.000,E1 273.498} C_DIS
LIN {X 0.012,Y -334.042,Z 1777.517,A 0.000,B 0.000,C 90.000,E1 273.037} C_DIS
LIN {X 0.149,Y -327.614,Z 1777.515,A 0.000,B 0.000,C 90.000,E1 272.579} C_DIS
LIN {X -0.133,Y -321.024,Z 1777.512,A 0.000,B 0.000,C 90.000,E1 272.236} C_DIS
LIN {X 0.146,Y -314.244,Z 1777.510,A 0.000,B 0.000,C 90.000,E1 271.835} C_DIS
LIN {X 0.062,Y -307.055,Z 1777.509,A 0.000,B 0.000,C 90.000,E1 271.547} C_DIS
LIN {X -0.009,Y -299.853,Z 1777.507,A 0.000,B 0.000,C 90.000,E1 271.318} C_DIS
LIN {X -0.022,Y -289.020,Z 1777.506,A 0.000,B 0.000,C 90.000,E1 271.031} C_DIS
LIN {X -0.125,Y -273.927,Z 1777.504,A 0.000,B 0.000,C 90.000,E1 270.745} C_DIS
LIN {X 0.041,Y -261.362,Z 1777.503,A 0.000,B 0.000,C 90.000,E1 270.516} C_DIS
LIN {X 0.089,Y -244.161,Z 1777.502,A 0.000,B 0.000,C 90.000,E1 270.344} C_DIS
LIN {X -0.101,Y -232.227,Z 1777.502,A 0.000,B 0.000,C 90.000,E1 270.344} C_DIS
LIN {X 0.071,Y -181.581,Z 1777.502,A 0.000,B 0.000,C 90.000,E1 270.286} C_DIS
LIN {X 0.022,Y -180.894,Z 1777.473,A 0.000,B 0.000,C 90.000,E1 265.179} C_DIS
LIN {X -0.078,Y -179.520,Z 1777.454,A 0.000,B 0.000,C 90.000,E1 261.837} C_DIS
LIN {X 0.084,Y -179.022,Z 1777.445,A 0.000,B 0.000,C 90.000,E1 260.095} C_DIS
LIN {X -0.031,Y -178.660,Z 1777.440,A 0.000,B 0.000,C 90.000,E1 259.285} C_DIS
LIN {X 0.075,Y -175.709,Z 1777.412,A 0.000,B 0.000,C 90.000,E1 254.157} C_DIS
LIN {X 0.086,Y -172.425,Z 1777.388,A 0.000,B 0.000,C 90.000,E1 249.880} C_DIS
LIN {X 0.102,Y -171.249,Z 1777.379,A 0.000,B 0.000,C 90.000,E1 248.156} C_DIS
LIN {X -0.074,Y -167.524,Z 1777.355,A 0.000,B 0.000,C 90.000,E1 243.896} C_DIS
LIN {X 0.009,Y -166.919,Z 1777.350,A 0.000,B 0.000,C 90.000,E1 242.999} C_DIS
LIN {X -0.077,Y -162.228,Z 1777.321,A 0.000,B 0.000,C 90.000,E1 237.788} C_DIS
LIN {X -0.020,Y -160.812,Z 1777.311,A 0.000,B 0.000,C 90.000,E1 236.008} C_DIS
LIN {X -0.042,Y -157.597,Z 1777.292,A 0.000,B 0.000,C 90.000,E1 232.477} C_DIS
LIN {X 0.016,Y -155.632,Z 1777.277,A 0.000,B 0.000,C 90.000,E1 229.784} C_DIS
LIN {X -0.049,Y -151.906,Z 1777.252,A 0.000,B 0.000,C 90.000,E1 225.324} C_DIS
LIN {X -0.033,Y -150.137,Z 1777.237,A 0.000,B 0.000,C 90.000,E1 222.609} C_DIS
LIN {X 0.003,Y -146.924,Z 1777.211,A 0.000,B 0.000,C 90.000,E1 218.051} C_DIS
LIN {X -0.004,Y -145.512,Z 1777.196,A 0.000,B 0.000,C 90.000,E1 215.311} C_DIS
LIN {X -0.010,Y -142.914,Z 1777.171,A 0.000,B 0.000,C 90.000,E1 210.718} C_DIS
LIN {X 0.042,Y -141.535,Z 1777.150,A 0.000,B 0.000,C 90.000,E1 207.001} C_DIS
LIN {X 0.086,Y -139.400,Z 1777.114,A 0.000,B 0.000,C 90.000,E1 200.482} C_DIS
LIN {X -0.040,Y -139.115,Z 1777.104,A 0.000,B 0.000,C 90.000,E1 198.671} C_DIS
LIN {X -0.009,Y -138.352,Z 1777.057,A 0.000,B 0.000,C 90.000,E1 190.254} C_DIS
LIN {X -0.018,Y -139.506,Z 1777.005,A 0.000,B 0.000,C 90.000,E1 180.917} C_DIS
LIN {X 0.063,Y -141.142,Z 1776.974,A 0.000,B 0.000,C 90.000,E1 175.298} C_DIS
LIN {X 0.016,Y -142.522,Z 1776.959,A 0.000,B 0.000,C 90.000,E1 172.534} C_DIS
LIN {X -0.038,Y -144.786,Z 1776.933,A 0.000,B 0.000,C 90.000,E1 167.937} C_DIS
LIN {X -0.050,Y -147.402,Z 1776.912,A 0.000,B 0.000,C 90.000,E1 164.267} C_DIS
LIN {X -0.020,Y -149.977,Z 1776.892,A 0.000,B 0.000,C 90.000,E1 160.604} C_DIS
LIN {X -0.011,Y -153.301,Z 1776.872,A 0.000,B 0.000,C 90.000,E1 156.975} C_DIS
LIN {X -0.023,Y -155.003,Z 1776.862,A 0.000,B 0.000,C 90.000,E1 155.177} C_DIS
LIN {X -0.011,Y -158.645,Z 1776.842,A 0.000,B 0.000,C 90.000,E1 151.591} C_DIS
LIN {X 0.010,Y -161.921,Z 1776.827,A 0.000,B 0.000,C 90.000,E1 148.918} C_DIS
LIN {X 0.033,Y -166.112,Z 1776.808,A 0.000,B 0.000,C 90.000,E1 145.388} C_DIS
LIN {X 0.031,Y -171.121,Z 1776.788,A 0.000,B 0.000,C 90.000,E1 141.904} C_DIS
LIN {X -0.050,Y -175.997,Z 1776.769,A 0.000,B 0.000,C 90.000,E1 138.485} C_DIS
LIN {X 0.063,Y -180.245,Z 1776.755,A 0.000,B 0.000,C 90.000,E1 135.891} C_DIS
LIN {X 0.037,Y -185.659,Z 1776.736,A 0.000,B 0.000,C 90.000,E1 132.528} C_DIS
LIN {X 0.090,Y -190.259,Z 1776.722,A 0.000,B 0.000,C 90.000,E1 130.011} C_DIS
LIN {X -0.020,Y -197.587,Z 1776.700,A 0.000,B 0.000,C 90.000,E1 125.931} C_DIS
LIN {X -0.095,Y -200.849,Z 1776.691,A 0.000,B 0.000,C 90.000,E1 124.326} C_DIS
LIN {X -0.011,Y -206.747,Z 1776.673,A 0.000,B 0.000,C 90.000,E1 121.082} C_DIS
LIN {X -0.025,Y -210.659,Z 1776.662,A 0.000,B 0.000,C 90.000,E1 119.155} C_DIS
LIN {X 0.111,Y -210.946,Z 1776.661,A 0.000,B 0.000,C 90.000,E1 118.949} C_DIS
LIN {X 0.134,Y -337.216,Z 1776.661,A 0.000,B 0.000,C 90.000,E1 118.949} C_DIS
LIN {X 0.043,Y -342.540,Z 1776.660,A 0.000,B 0.000,C 90.000,E1 118.821} C_DIS
LIN {X -0.005,Y -344.767,Z 1776.659,A 0.000,B 0.000,C 90.000,E1 118.693} C_DIS
LIN {X 0.099,Y -348.627,Z 1776.657,A 0.000,B 0.000,C 90.000,E1 118.309} C_DIS
LIN {X 0.173,Y -352.052,Z 1776.654,A 0.000,B 0.000,C 90.000,E1 117.769} C_DIS
LIN {X 0.135,Y -366.867,Z 1776.638,A 0.000,B 0.000,C 90.000,E1 114.771} C_DIS
LIN {X 0.001,Y -381.798,Z 1776.623,A 0.000,B 0.000,C 90.000,E1 112.153} C_DIS
LIN {X 0.178,Y -399.987,Z 1776.607,A 0.000,B 0.000,C 90.000,E1 109.268} C_DIS
LIN {X -0.106,Y -417.188,Z 1776.593,A 0.000,B 0.000,C 90.000,E1 106.804} C_DIS
LIN {X 0.188,Y -432.938,Z 1776.581,A 0.000,B 0.000,C 90.000,E1 104.592} C_DIS
LIN {X 0.100,Y -444.812,Z 1776.572,A 0.000,B 0.000,C 90.000,E1 103.008} C_DIS
LIN {X -0.027,Y -454.486,Z 1776.565,A 0.000,B 0.000,C 90.000,E1 101.715} C_DIS
LIN {X 0.143,Y -461.803,Z 1776.559,A 0.000,B 0.000,C 90.000,E1 100.658} C_DIS
LIN {X 0.012,Y -466.757,Z 1776.555,A 0.000,B 0.000,C 90.000,E1 99.905} C_DIS
LIN {X 0.159,Y -469.569,Z 1776.552,A 0.000,B 0.000,C 90.000,E1 99.378} C_DIS
LIN {X -0.068,Y -470.727,Z 1776.551,A 0.000,B 0.000,C 90.000,E1 99.151} C_DIS
LIN {X -0.220,Y -471.621,Z 1776.549,A 0.000,B 0.000,C 90.000,E1 98.916} C_DIS
LIN {X -0.116,Y -472.024,Z 1776.547,A 0.000,B 0.000,C 90.000,E1 98.398} C_DIS
LIN {X -0.236,Y -472.408,Z 1776.513,A 0.000,B 0.000,C 90.000,E1 92.350} C_DIS
LIN {X -0.148,Y -472.329,Z 1776.510,A 0.000,B 0.000,C 90.000,E1 91.835} C_DIS
LIN {X -0.045,Y -471.144,Z 1776.507,A 0.000,B 0.000,C 90.000,E1 91.318} C_DIS
LIN {X 0.042,Y -469.443,Z 1776.505,A 0.000,B 0.000,C 90.000,E1 90.802} C_DIS
LIN {X -0.072,Y -466.376,Z 1776.500,A 0.000,B 0.000,C 90.000,E1 90.057} C_DIS
LIN {X 0.038,Y -461.665,Z 1776.495,A 0.000,B 0.000,C 90.000,E1 89.026} C_DIS
LIN {X -0.120,Y -455.184,Z 1776.488,A 0.000,B 0.000,C 90.000,E1 87.764} C_DIS
LIN {X 0.081,Y -448.288,Z 1776.480,A 0.000,B 0.000,C 90.000,E1 86.445} C_DIS
LIN {X 0.210,Y -441.024,Z 1776.473,A 0.000,B 0.000,C 90.000,E1 85.122} C_DIS
LIN {X 0.126,Y -430.520,Z 1776.463,A 0.000,B 0.000,C 90.000,E1 83.280} C_DIS
LIN {X -0.117,Y -419.771,Z 1776.452,A 0.000,B 0.000,C 90.000,E1 81.432} C_DIS
LIN {X -0.039,Y -408.968,Z 1776.442,A 0.000,B 0.000,C 90.000,E1 79.511} C_DIS
LIN {X -0.011,Y -396.769,Z 1776.429,A 0.000,B 0.000,C 90.000,E1 77.285} C_DIS
LIN {X -0.183,Y -384.641,Z 1776.417,A 0.000,B 0.000,C 90.000,E1 75.046} C_DIS
LIN {X 0.012,Y -369.815,Z 1776.401,A 0.000,B 0.000,C 90.000,E1 72.127} C_DIS
LIN {X 0.025,Y -359.793,Z 1776.389,A 0.000,B 0.000,C 90.000,E1 70.061} C_DIS
LIN {X 0.019,Y -347.205,Z 1776.374,A 0.000,B 0.000,C 90.000,E1 67.358} C_DIS
LIN {X 0.079,Y -335.019,Z 1776.359,A 0.000,B 0.000,C 90.000,E1 64.588} C_DIS
LIN {X 0.036,Y -325.759,Z 1776.347,A 0.000,B 0.000,C 90.000,E1 62.410} C_DIS
LIN {X -0.065,Y -319.003,Z 1776.338,A 0.000,B 0.000,C 90.000,E1 60.845} C_DIS
LIN {X -0.048,Y -310.469,Z 1776.327,A 0.000,B 0.000,C 90.000,E1 58.918} C_DIS
LIN {X -0.031,Y -301.628,Z 1776.316,A 0.000,B 0.000,C 90.000,E1 56.962} C_DIS
LIN {X 0.141,Y -291.092,Z 1776.304,A 0.000,B 0.000,C 90.000,E1 54.609} C_DIS
LIN {X -0.020,Y -276.729,Z 1776.285,A 0.000,B 0.000,C 90.000,E1 51.251} C_DIS
LIN {X -0.003,Y -264.565,Z 1776.267,A 0.000,B 0.000,C 90.000,E1 48.119} C_DIS
LIN {X -0.031,Y -254.318,Z 1776.252,A 0.000,B 0.000,C 90.000,E1 45.283} C_DIS
LIN {X 0.044,Y -243.134,Z 1776.233,A 0.000,B 0.000,C 90.000,E1 42.000} C_DIS
LIN {X 0.015,Y -232.600,Z 1776.215,A 0.000,B 0.000,C 90.000,E1 38.669} C_DIS
LIN {X 0.003,Y -223.770,Z 1776.198,A 0.000,B 0.000,C 90.000,E1 35.644} C_DIS
LIN {X 0.086,Y -215.496,Z 1776.181,A 0.000,B 0.000,C 90.000,E1 32.546} C_DIS
LIN {X 0.102,Y -207.770,Z 1776.164,A 0.000,B 0.000,C 90.000,E1 29.411} C_DIS
LIN {X 0.088,Y -200.805,Z 1776.146,A 0.000,B 0.000,C 90.000,E1 26.232} C_DIS
LIN {X 0.005,Y -194.580,Z 1776.128,A 0.000,B 0.000,C 90.000,E1 23.025} C_DIS
LIN {X -0.016,Y -189.182,Z 1776.110,A 0.000,B 0.000,C 90.000,E1 19.758} C_DIS
LIN {X -0.005,Y -184.737,Z 1776.091,A 0.000,B 0.000,C 90.000,E1 16.441} C_DIS
LIN {X -0.079,Y -181.205,Z 1776.073,A 0.000,B 0.000,C 90.000,E1 13.119} C_DIS
LIN {X 0.049,Y -177.834,Z 1776.049,A 0.000,B 0.000,C 90.000,E1 8.859} C_DIS
LIN {X -0.034,Y -175.109,Z 1776.021,A 0.000,B 0.000,C 90.000,E1 3.784} C_DIS
LIN {X 0.007,Y -173.678,Z 1775.978,A 0.000,B 0.000,C 90.000,E1 356.102} C_DIS
LIN {X 0.031,Y -174.178,Z 1775.945,A 0.000,B 0.000,C 90.000,E1 350.095} C_DIS
LIN {X -0.011,Y -176.319,Z 1775.907,A 0.000,B 0.000,C 90.000,E1 343.268} C_DIS
LIN {X 0.015,Y -179.323,Z 1775.879,A 0.000,B 0.000,C 90.000,E1 338.156} C_DIS
LIN {X 0.059,Y -183.210,Z 1775.851,A 0.000,B 0.000,C 90.000,E1 333.076} C_DIS
LIN {X -0.026,Y -187.470,Z 1775.827,A 0.000,B 0.000,C 90.000,E1 328.918} C_DIS
LIN {X -0.009,Y -191.613,Z 1775.809,A 0.000,B 0.000,C 90.000,E1 325.595} C_DIS
LIN {X -0.034,Y -196.701,Z 1775.791,A 0.000,B 0.000,C 90.000,E1 322.316} C_DIS
LIN {X 0.003,Y -202.856,Z 1775.773,A 0.000,B 0.000,C 90.000,E1 319.057} C_DIS
LIN {X -0.136,Y -210.364,Z 1775.755,A 0.000,B 0.000,C 90.000,E1 315.891} C_DIS
LIN {X -0.032,Y -216.903,Z 1775.742,A 0.000,B 0.000,C 90.000,E1 313.500} C_DIS
LIN {X 0.060,Y -221.906,Z 1775.733,A 0.000,B 0.000,C 90.000,E1 311.919} C_DIS
LIN {X 0.065,Y -227.552,Z 1775.724,A 0.000,B 0.000,C 90.000,E1 310.378} C_DIS
LIN {X 0.130,Y -235.608,Z 1775.714,A 0.000,B 0.000,C 90.000,E1 308.463} C_DIS
LIN {X -0.017,Y -244.815,Z 1775.703,A 0.000,B 0.000,C 90.000,E1 306.629} C_DIS
LIN {X -0.115,Y -254.959,Z 1775.693,A 0.000,B 0.000,C 90.000,E1 304.818} C_DIS
LIN {X 0.045,Y -272.885,Z 1775.677,A 0.000,B 0.000,C 90.000,E1 301.926} C_DIS
LIN {X -0.139,Y -292.442,Z 1775.662,A 0.000,B 0.000,C 90.000,E1 299.205} C_DIS
LIN {X 0.167,Y -313.174,Z 1775.647,A 0.000,B 0.000,C 90.000,E1 296.488} C_DIS
LIN {X 0.043,Y -326.502,Z 1775.638,A 0.000,B 0.000,C 90.000,E1 294.899} C_DIS
LIN {X 0.054,Y -339.555,Z 1775.630,A 0.000,B 0.000,C 90.000,E1 293.334} C_DIS
LIN {X 0.063,Y -349.746,Z 1775.623,A 0.000,B 0.000,C 90.000,E1 292.099} C_DIS
LIN {X -0.144,Y -359.641,Z 1775.616,A 0.000,B 0.000,C 90.000,E1 290.918} C_DIS
LIN {X -0.037,Y -364.416,Z 1775.613,A 0.000,B 0.000,C 90.000,E1 290.301} C_DIS
LIN {X 0.055,Y -371.032,Z 1775.608,A 0.000,B 0.000,C 90.000,E1 289.396} C_DIS
LIN {X -0.135,Y -376.847,Z 1775.603,A 0.000,B 0.000,C 90.000,E1 288.544} C_DIS
LIN {X 0.080,Y -381.733,Z 1775.598,A 0.000,B 0.000,C 90.000,E1 287.638} C_DIS
LIN {X -0.151,Y -384.465,Z 1775.595,A 0.000,B 0.000,C 90.000,E1 287.094} C_DIS
LIN {X 0.001,Y -386.767,Z 1775.592,A 0.000,B 0.000,C 90.000,E1 286.496} C_DIS
LIN {X 0.170,Y -388.713,Z 1775.589,A 0.000,B 0.000,C 90.000,E1 285.898} C_DIS
LIN {X -0.134,Y -390.298,Z 1775.585,A 0.000,B 0.000,C 90.000,E1 285.371} C_DIS
LIN {X 0.054,Y -391.554,Z 1775.582,A 0.000,B 0.000,C 90.000,E1 284.773} C_DIS
LIN {X -0.226,Y -392.426,Z 1775.579,A 0.000,B 0.000,C 90.000,E1 284.245} C_DIS
LIN {X -0.024,Y -392.954,Z 1775.576,A 0.000,B 0.000,C 90.000,E1 283.647} C_DIS
LIN {X 0.092,Y -393.099,Z 1775.573,A 0.000,B 0.000,C 90.000,E1 283.063} C_DIS
LIN {X -0.171,Y -392.899,Z 1775.569,A 0.000,B 0.000,C 90.000,E1 282.535} C_DIS
LIN {X -0.049,Y -392.329,Z 1775.566,A 0.000,B 0.000,C 90.000,E1 281.951} C_DIS
LIN {X 0.074,Y -391.418,Z 1775.563,A 0.000,B 0.000,C 90.000,E1 281.366} C_DIS
LIN {X -0.193,Y -390.118,Z 1775.560,A 0.000,B 0.000,C 90.000,E1 280.838} C_DIS
LIN {X -0.081,Y -388.467,Z 1775.557,A 0.000,B 0.000,C 90.000,E1 280.254} C_DIS
LIN {X 0.064,Y -385.275,Z 1775.552,A 0.000,B 0.000,C 90.000,E1 279.378} C_DIS
LIN {X 0.116,Y -381.277,Z 1775.547,A 0.000,B 0.000,C 90.000,E1 278.511} C_DIS
LIN {X 0.128,Y -376.633,Z 1775.543,A 0.000,B 0.000,C 90.000,E1 277.644} C_DIS
LIN {X 0.105,Y -371.263,Z 1775.538,A 0.000,B 0.000,C 90.000,E1 276.777} C_DIS
LIN {X 0.048,Y -367.091,Z 1775.535,A 0.000,B 0.000,C 90.000,E1 276.201} C_DIS
LIN {X -0.031,Y -362.391,Z 1775.531,A 0.000,B 0.000,C 90.000,E1 275.625} C_DIS
LIN {X -0.133,Y -357.078,Z 1775.528,A 0.000,B 0.000,C 90.000,E1 275.049} C_DIS
LIN {X -0.159,Y -351.205,Z 1775.525,A 0.000,B 0.000,C 90.000,E1 274.473} C_DIS
LIN {X 0.118,Y -345.251,Z 1775.522,A 0.000,B 0.000,C 90.000,E1 273.898} C_DIS
LIN {X -0.092,Y -339.234,Z 1775.519,A 0.000,B 0.000,C 90.000,E1 273.440} C_DIS
LIN {X 0.008,Y -329.864,Z 1775.515,A 0.000,B 0.000,C 90.000,E1 272.751} C_DIS
LIN {X 0.009,Y -323.455,Z 1775.513,A 0.000,B 0.000,C 90.000,E1 272.350} C_DIS
LIN {X -0.108,Y -316.746,Z 1775.511,A 0.000,B 0.000,C 90.000,E1 272.007} C_DIS
LIN {X 0.012,Y -309.689,Z 1775.509,A 0.000,B 0.000,C 90.000,E1 271.661} C_DIS
LIN {X 0.098,Y -302.229,Z 1775.508,A 0.000,B 0.000,C 90.000,E1 271.375} C_DIS
LIN {X -0.034,Y -291.117,Z 1775.506,A 0.000,B 0.000,C 90.000,E1 271.088} C_DIS
LIN {X -0.084,Y -280.004,Z 1775.505,A 0.000,B 0.000,C 90.000,E1 270.859} C_DIS
LIN {X 0.006,Y -267.991,Z 1775.504,A 0.000,B 0.000,C 90.000,E1 270.630} C_DIS
LIN {X -0.030,Y -258.902,Z 1775.503,A 0.000,B 0.000,C 90.000,E1 270.516} C_DIS
LIN {X -0.102,Y -243.714,Z 1775.502,A 0.000,B 0.000,C 90.000,E1 270.401} C_DIS
LIN {X -0.029,Y -233.725,Z 1775.502,A 0.000,B 0.000,C 90.000,E1 270.344} C_DIS
LIN {X -0.041,Y -181.580,Z 1775.502,A 0.000,B 0.000,C 90.000,E1 270.344} C_DIS
LIN {X 0.042,Y -180.901,Z 1775.474,A 0.000,B 0.000,C 90.000,E1 265.241} C_DIS
LIN {X -0.008,Y -180.223,Z 1775.464,A 0.000,B 0.000,C 90.000,E1 263.571} C_DIS
LIN {X -0.055,Y -179.039,Z 1775.446,A 0.000,B 0.000,C 90.000,E1 260.208} C_DIS
LIN {X 0.008,Y -178.704,Z 1775.441,A 0.000,B 0.000,C 90.000,E1 259.342} C_DIS
LIN {X -0.051,Y -175.753,Z 1775.412,A 0.000,B 0.000,C 90.000,E1 254.267} C_DIS
LIN {X -0.048,Y -171.936,Z 1775.384,A 0.000,B 0.000,C 90.000,E1 249.135} C_DIS
LIN {X -0.072,Y -171.317,Z 1775.379,A 0.000,B 0.000,C 90.000,E1 248.284} C_DIS
LIN {X -0.019,Y -167.575,Z 1775.355,A 0.000,B 0.000,C 90.000,E1 243.948} C_DIS
LIN {X -0.080,Y -166.207,Z 1775.346,A 0.000,B 0.000,C 90.000,E1 242.231} C_DIS
LIN {X -0.090,Y -162.972,Z 1775.326,A 0.000,B 0.000,C 90.000,E1 238.742} C_DIS
LIN {X -0.042,Y -160.885,Z 1775.312,A 0.000,B 0.000,C 90.000,E1 236.087} C_DIS
LIN {X -0.064,Y -157.655,Z 1775.292,A 0.000,B 0.000,C 90.000,E1 232.557} C_DIS
LIN {X 0.094,Y -155.692,Z 1775.277,A 0.000,B 0.000,C 90.000,E1 229.828} C_DIS
LIN {X -0.070,Y -151.957,Z 1775.252,A 0.000,B 0.000,C 90.000,E1 225.405} C_DIS
LIN {X -0.053,Y -150.197,Z 1775.237,A 0.000,B 0.000,C 90.000,E1 222.690} C_DIS
LIN {X 0.077,Y -146.967,Z 1775.212,A 0.000,B 0.000,C 90.000,E1 218.096} C_DIS
LIN {X -0.019,Y -145.554,Z 1775.197,A 0.000,B 0.000,C 90.000,E1 215.391} C_DIS
LIN {X -0.020,Y -142.947,Z 1775.171,A 0.000,B 0.000,C 90.000,E1 210.797} C_DIS
LIN {X 0.037,Y -141.573,Z 1775.151,A 0.000,B 0.000,C 90.000,E1 207.078} C_DIS
LIN {X -0.041,Y -139.413,Z 1775.114,A 0.000,B 0.000,C 90.000,E1 200.610} C_DIS
LIN {X 0.012,Y -139.136,Z 1775.104,A 0.000,B 0.000,C 90.000,E1 198.725} C_DIS
LIN {X 0.039,Y -138.349,Z 1775.057,A 0.000,B 0.000,C 90.000,E1 190.310} C_DIS
LIN {X 0.026,Y -139.495,Z 1775.005,A 0.000,B 0.000,C 90.000,E1 180.974} C_DIS
LIN {X -0.033,Y -141.110,Z 1774.974,A 0.000,B 0.000,C 90.000,E1 175.412} C_DIS
LIN {X 0.061,Y -142.489,Z 1774.959,A 0.000,B 0.000,C 90.000,E1 172.591} C_DIS
LIN {X 0.009,Y -144.740,Z 1774.933,A 0.000,B 0.000,C 90.000,E1 167.993} C_DIS
LIN {X -0.041,Y -147.347,Z 1774.913,A 0.000,B 0.000,C 90.000,E1 164.338} C_DIS
LIN {X 0.023,Y -150.671,Z 1774.888,A 0.000,B 0.000,C 90.000,E1 159.752} C_DIS
LIN {X -0.096,Y -154.151,Z 1774.867,A 0.000,B 0.000,C 90.000,E1 156.177} C_DIS
LIN {X 0.039,Y -157.580,Z 1774.848,A 0.000,B 0.000,C 90.000,E1 152.538} C_DIS
LIN {X -0.010,Y -161.828,Z 1774.828,A 0.000,B 0.000,C 90.000,E1 148.997} C_DIS
LIN {X 0.008,Y -166.019,Z 1774.808,A 0.000,B 0.000,C 90.000,E1 145.468} C_DIS
LIN {X 0.001,Y -171.019,Z 1774.789,A 0.000,B 0.000,C 90.000,E1 141.984} C_DIS
LIN {X 0.032,Y -175.889,Z 1774.770,A 0.000,B 0.000,C 90.000,E1 138.528} C_DIS
LIN {X -0.092,Y -181.494,Z 1774.751,A 0.000,B 0.000,C 90.000,E1 135.162} C_DIS
LIN {X 0.044,Y -187.010,Z 1774.732,A 0.000,B 0.000,C 90.000,E1 131.757} C_DIS
LIN {X 0.045,Y -190.128,Z 1774.723,A 0.000,B 0.000,C 90.000,E1 130.092} C_DIS
LIN {X 0.064,Y -195.899,Z 1774.704,A 0.000,B 0.000,C 90.000,E1 126.790} C_DIS
LIN {X 0.021,Y -200.729,Z 1774.691,A 0.000,B 0.000,C 90.000,E1 124.358} C_DIS
LIN {X 0.047,Y -206.617,Z 1774.673,A 0.000,B 0.000,C 90.000,E1 121.131} C_DIS
LIN {X -0.004,Y -210.696,Z 1774.662,A 0.000,B 0.000,C 90.000,E1 119.127} C_DIS
LIN {X -0.018,Y -210.921,Z 1774.661,A 0.000,B 0.000,C 90.000,E1 118.999} C_DIS
LIN {X -0.065,Y -337.615,Z 1774.661,A 0.000,B 0.000,C 90.000,E1 118.999} C_DIS
LIN {X 0.159,Y -338.572,Z 1774.661,A 0.000,B 0.000,C 90.000,E1 118.949} C_DIS
LIN {X 0.078,Y -344.010,Z 1774.660,A 0.000,B 0.000,C 90.000,E1 118.743} C_DIS
LIN {X 0.107,Y -347.066,Z 1774.658,A 0.000,B 0.000,C 90.000,E1 118.487} C_DIS
LIN {X 0.048,Y -350.731,Z 1774.656,A 0.000,B 0.000,C 90.000,E1 118.025} C_DIS
LIN {X -0.078,Y -353.787,Z 1774.652,A 0.000,B 0.000,C 90.000,E1 117.436} C_DIS
LIN {X 0.041,Y -367.198,Z 1774.637,A 0.000,B 0.000,C 90.000,E1 114.719} C_DIS
LIN {X 0.057,Y -382.175,Z 1774.623,A 0.000,B 0.000,C 90.000,E1 112.078} C_DIS
LIN {X 0.107,Y -400.730,Z 1774.607,A 0.000,B 0.000,C 90.000,E1 109.214} C_DIS
LIN {X -0.025,Y -418.504,Z 1774.593,A 0.000,B 0.000,C 90.000,E1 106.732} C_DIS
LIN {X 0.189,Y -434.867,Z 1774.581,A 0.000,B 0.000,C 90.000,E1 104.537} C_DIS
LIN {X 0.032,Y -449.406,Z 1774.571,A 0.000,B 0.000,C 90.000,E1 102.703} C_DIS
LIN {X 0.142,Y -461.717,Z 1774.562,A 0.000,B 0.000,C 90.000,E1 101.130} C_DIS
LIN {X -0.143,Y -469.580,Z 1774.556,A 0.000,B 0.000,C 90.000,E1 100.141} C_DIS
LIN {X -0.124,Y -475.065,Z 1774.552,A 0.000,B 0.000,C 90.000,E1 99.378} C_DIS
LIN {X -0.143,Y -479.858,Z 1774.548,A 0.000,B 0.000,C 90.000,E1 98.624} C_DIS
LIN {X 0.007,Y -482.295,Z 1774.545,A 0.000,B 0.000,C 90.000,E1 98.106} C_DIS
LIN {X 0.176,Y -483.282,Z 1774.542,A 0.000,B 0.000,C 90.000,E1 97.587} C_DIS
LIN {X 0.140,Y -483.375,Z 1774.520,A 0.000,B 0.000,C 90.000,E1 93.612} C_DIS
LIN {X -0.167,Y -482.856,Z 1774.517,A 0.000,B 0.000,C 90.000,E1 93.151} C_DIS
LIN {X -0.018,Y -481.412,Z 1774.515,A 0.000,B 0.000,C 90.000,E1 92.636} C_DIS
LIN {X 0.131,Y -479.555,Z 1774.512,A 0.000,B 0.000,C 90.000,E1 92.121} C_DIS
LIN {X -0.060,Y -475.161,Z 1774.506,A 0.000,B 0.000,C 90.000,E1 91.146} C_DIS
LIN {X -0.041,Y -468.972,Z 1774.499,A 0.000,B 0.000,C 90.000,E1 89.885} C_DIS
LIN {X -0.109,Y -462.216,Z 1774.492,A 0.000,B 0.000,C 90.000,E1 88.625} C_DIS
LIN {X -0.035,Y -453.640,Z 1774.484,A 0.000,B 0.000,C 90.000,E1 87.078} C_DIS
LIN {X -0.085,Y -444.669,Z 1774.475,A 0.000,B 0.000,C 90.000,E1 85.527} C_DIS
LIN {X -0.094,Y -433.790,Z 1774.465,A 0.000,B 0.000,C 90.000,E1 83.685} C_DIS
LIN {X 0.150,Y -422.718,Z 1774.454,A 0.000,B 0.000,C 90.000,E1 81.781} C_DIS
LIN {X -0.127,Y -411.588,Z 1774.444,A 0.000,B 0.000,C 90.000,E1 79.916} C_DIS
LIN {X -0.118,Y -398.984,Z 1774.432,A 0.000,B 0.000,C 90.000,E1 77.701} C_DIS
LIN {X 0.132,Y -386.499,Z 1774.419,A 0.000,B 0.000,C 90.000,E1 75.408} C_DIS
LIN {X 0.011,Y -371.521,Z 1774.403,A 0.000,B 0.000,C 90.000,E1 72.543} C_DIS
LIN {X 0.012,Y -360.021,Z 1774.390,A 0.000,B 0.000,C 90.000,E1 70.188} C_DIS
LIN {X -0.021,Y -348.767,Z 1774.377,A 0.000,B 0.000,C 90.000,E1 67.794} C_DIS
LIN {X -0.060,Y -336.505,Z 1774.361,A 0.000,B 0.000,C 90.000,E1 65.049} C_DIS
LIN {X -0.076,Y -327.215,Z 1774.349,A 0.000,B 0.000,C 90.000,E1 62.871} C_DIS
LIN {X -0.066,Y -319.147,Z 1774.339,A 0.000,B 0.000,C 90.000,E1 60.973} C_DIS
LIN {X -0.205,Y -310.679,Z 1774.328,A 0.000,B 0.000,C 90.000,E1 59.076} C_DIS
LIN {X -0.021,Y -301.870,Z 1774.317,A 0.000,B 0.000,C 90.000,E1 57.089} C_DIS
LIN {X -0.004,Y -292.832,Z 1774.306,A 0.000,B 0.000,C 90.000,E1 55.102} C_DIS
LIN {X -0.002,Y -279.769,Z 1774.289,A 0.000,B 0.000,C 90.000,E1 52.065} C_DIS
LIN {X 0.015,Y -268.760,Z 1774.274,A 0.000,B 0.000,C 90.000,E1 49.299} C_DIS
LIN {X -0.036,Y -257.058,Z 1774.256,A 0.000,B 0.000,C 90.000,E1 46.134} C_DIS
LIN {X 0.113,Y -245.700,Z 1774.238,A 0.000,B 0.000,C 90.000,E1 42.852} C_DIS
LIN {X -0.029,Y -234.963,Z 1774.220,A 0.000,B 0.000,C 90.000,E1 39.564} C_DIS
LIN {X -0.029,Y -224.862,Z 1774.201,A 0.000,B 0.000,C 90.000,E1 36.171} C_DIS
LIN {X 0.030,Y -216.528,Z 1774.184,A 0.000,B 0.000,C 90.000,E1 33.086} C_DIS
LIN {X -0.109,Y -208.690,Z 1774.167,A 0.000,B 0.000,C 90.000,E1 30.001} C_DIS
LIN {X -0.001,Y -201.608,Z 1774.149,A 0.000,B 0.000,C 90.000,E1 26.796} C_DIS
LIN {X 0.014,Y -195.263,Z 1774.131,A 0.000,B 0.000,C 90.000,E1 23.567} C_DIS
LIN {X 0.002,Y -189.730,Z 1774.113,A 0.000,B 0.000,C 90.000,E1 20.301} C_DIS
LIN {X 0.026,Y -185.123,Z 1774.094,A 0.000,B 0.000,C 90.000,E1 16.985} C_DIS
LIN {X 0.007,Y -181.446,Z 1774.076,A 0.000,B 0.000,C 90.000,E1 13.647} C_DIS
LIN {X -0.033,Y -177.948,Z 1774.052,A 0.000,B 0.000,C 90.000,E1 9.443} C_DIS
LIN {X -0.087,Y -175.043,Z 1774.024,A 0.000,B 0.000,C 90.000,E1 4.359} C_DIS
LIN {X 0.002,Y -173.417,Z 1773.978,A 0.000,B 0.000,C 90.000,E1 356.102} C_DIS
LIN {X 0.013,Y -173.895,Z 1773.945,A 0.000,B 0.000,C 90.000,E1 350.095} C_DIS
LIN {X -0.043,Y -176.043,Z 1773.907,A 0.000,B 0.000,C 90.000,E1 343.268} C_DIS
LIN {X -0.028,Y -179.066,Z 1773.879,A 0.000,B 0.000,C 90.000,E1 338.156} C_DIS
LIN {X 0.008,Y -183.024,Z 1773.850,A 0.000,B 0.000,C 90.000,E1 333.076} C_DIS
LIN {X 0.075,Y -187.303,Z 1773.827,A 0.000,B 0.000,C 90.000,E1 328.869} C_DIS
LIN {X -0.073,Y -191.529,Z 1773.809,A 0.000,B 0.000,C 90.000,E1 325.595} C_DIS
LIN {X 0.053,Y -196.675,Z 1773.791,A 0.000,B 0.000,C 90.000,E1 322.271} C_DIS
LIN {X 0.086,Y -202.892,Z 1773.772,A 0.000,B 0.000,C 90.000,E1 319.013} C_DIS
LIN {X 0.090,Y -210.475,Z 1773.755,A 0.000,B 0.000,C 90.000,E1 315.810} C_DIS
LIN {X 0.044,Y -217.041,Z 1773.741,A 0.000,B 0.000,C 90.000,E1 313.461} C_DIS
LIN {X 0.060,Y -223.440,Z 1773.731,A 0.000,B 0.000,C 90.000,E1 311.515} C_DIS
LIN {X -0.066,Y -229.280,Z 1773.722,A 0.000,B 0.000,C 90.000,E1 310.011} C_DIS
LIN {X 0.060,Y -235.823,Z 1773.714,A 0.000,B 0.000,C 90.000,E1 308.463} C_DIS
LIN {X 0.110,Y -245.063,Z 1773.703,A 0.000,B 0.000,C 90.000,E1 306.583} C_DIS
LIN {X -0.051,Y -253.128,Z 1773.695,A 0.000,B 0.000,C 90.000,E1 305.152} C_DIS
LIN {X 0.059,Y -270.908,Z 1773.679,A 0.000,B 0.000,C 90.000,E1 302.260} C_DIS
LIN {X 0.076,Y -290.300,Z 1773.664,A 0.000,B 0.000,C 90.000,E1 299.489} C_DIS
LIN {X -0.087,Y -308.293,Z 1773.651,A 0.000,B 0.000,C 90.000,E1 297.180} C_DIS
LIN {X 0.109,Y -324.182,Z 1773.640,A 0.000,B 0.000,C 90.000,E1 295.207} C_DIS
LIN {X 0.138,Y -337.192,Z 1773.631,A 0.000,B 0.000,C 90.000,E1 293.643} C_DIS
LIN {X 0.106,Y -347.520,Z 1773.625,A 0.000,B 0.000,C 90.000,E1 292.408} C_DIS
LIN {X -0.078,Y -359.932,Z 1773.616,A 0.000,B 0.000,C 90.000,E1 290.918} C_DIS
LIN {X 0.032,Y -364.726,Z 1773.613,A 0.000,B 0.000,C 90.000,E1 290.301} C_DIS
LIN {X 0.127,Y -371.354,Z 1773.608,A 0.000,B 0.000,C 90.000,E1 289.396} C_DIS
LIN {X -0.059,Y -377.183,Z 1773.603,A 0.000,B 0.000,C 90.000,E1 288.544} C_DIS
LIN {X 0.161,Y -382.065,Z 1773.598,A 0.000,B 0.000,C 90.000,E1 287.638} C_DIS
LIN {X -0.069,Y -384.790,Z 1773.595,A 0.000,B 0.000,C 90.000,E1 287.094} C_DIS
LIN {X 0.086,Y -387.110,Z 1773.592,A 0.000,B 0.000,C 90.000,E1 286.496} C_DIS
LIN {X -0.116,Y -389.046,Z 1773.589,A 0.000,B 0.000,C 90.000,E1 285.953} C_DIS
LIN {X -0.043,Y -390.649,Z 1773.585,A 0.000,B 0.000,C 90.000,E1 285.371} C_DIS
LIN {X 0.147,Y -391.893,Z 1773.582,A 0.000,B 0.000,C 90.000,E1 284.773} C_DIS
LIN {X -0.132,Y -392.774,Z 1773.579,A 0.000,B 0.000,C 90.000,E1 284.245} C_DIS
LIN {X 0.074,Y -393.293,Z 1773.576,A 0.000,B 0.000,C 90.000,E1 283.647} C_DIS
LIN {X -0.192,Y -393.463,Z 1773.573,A 0.000,B 0.000,C 90.000,E1 283.119} C_DIS
LIN {X -0.071,Y -393.251,Z 1773.570,A 0.000,B 0.000,C 90.000,E1 282.535} C_DIS
LIN {X 0.055,Y -392.697,Z 1773.566,A 0.000,B 0.000,C 90.000,E1 281.951} C_DIS
LIN {X -0.206,Y -391.790,Z 1773.563,A 0.000,B 0.000,C 90.000,E1 281.422} C_DIS
LIN {X -0.086,Y -390.480,Z 1773.560,A 0.000,B 0.000,C 90.000,E1 280.838} C_DIS
LIN {X 0.028,Y -388.779,Z 1773.557,A 0.000,B 0.000,C 90.000,E1 280.254} C_DIS
LIN {X 0.131,Y -386.724,Z 1773.554,A 0.000,B 0.000,C 90.000,E1 279.670} C_DIS
LIN {X -0.184,Y -382.946,Z 1773.549,A 0.000,B 0.000,C 90.000,E1 278.859} C_DIS
LIN {X -0.132,Y -376.872,Z 1773.543,A 0.000,B 0.000,C 90.000,E1 277.701} C_DIS
LIN {X -0.150,Y -371.504,Z 1773.538,A 0.000,B 0.000,C 90.000,E1 276.834} C_DIS
LIN {X 0.161,Y -367.405,Z 1773.535,A 0.000,B 0.000,C 90.000,E1 276.201} C_DIS
LIN {X 0.083,Y -362.684,Z 1773.531,A 0.000,B 0.000,C 90.000,E1 275.625} C_DIS
LIN {X -0.020,Y -357.375,Z 1773.528,A 0.000,B 0.000,C 90.000,E1 275.049} C_DIS
LIN {X 0.108,Y -348.658,Z 1773.523,A 0.000,B 0.000,C 90.000,E1 274.188} C_DIS
LIN {X 0.085,Y -339.643,Z 1773.519,A 0.000,B 0.000,C 90.000,E1 273.440} C_DIS
LIN {X -0.142,Y -330.334,Z 1773.516,A 0.000,B 0.000,C 90.000,E1 272.808} C_DIS
LIN {X -0.132,Y -323.941,Z 1773.513,A 0.000,B 0.000,C 90.000,E1 272.407} C_DIS
LIN {X 0.061,Y -317.281,Z 1773.511,A 0.000,B 0.000,C 90.000,E1 272.007} C_DIS
LIN {X -0.143,Y -310.306,Z 1773.509,A 0.000,B 0.000,C 90.000,E1 271.718} C_DIS
LIN {X -0.053,Y -302.950,Z 1773.508,A 0.000,B 0.000,C 90.000,E1 271.432} C_DIS
LIN {X 0.086,Y -291.858,Z 1773.506,A 0.000,B 0.000,C 90.000,E1 271.088} C_DIS
LIN {X 0.027,Y -280.790,Z 1773.505,A 0.000,B 0.000,C 90.000,E1 270.859} C_DIS
LIN {X -0.132,Y -269.090,Z 1773.504,A 0.000,B 0.000,C 90.000,E1 270.688} C_DIS
LIN {X 0.108,Y -254.901,Z 1773.503,A 0.000,B 0.000,C 90.000,E1 270.458} C_DIS
LIN {X -0.075,Y -242.399,Z 1773.502,A 0.000,B 0.000,C 90.000,E1 270.401} C_DIS
LIN {X 0.030,Y -233.825,Z 1773.502,A 0.000,B 0.000,C 90.000,E1 270.344} C_DIS
LIN {X 0.004,Y -181.579,Z 1773.502,A 0.000,B 0.000,C 90.000,E1 270.344} C_DIS
LIN {X -0.025,Y -180.848,Z 1773.472,A 0.000,B 0.000,C 90.000,E1 264.951} C_DIS
LIN {X 0.058,Y -178.958,Z 1773.444,A 0.000,B 0.000,C 90.000,E1 259.859} C_DIS
LIN {X -0.050,Y -177.361,Z 1773.430,A 0.000,B 0.000,C 90.000,E1 257.353} C_DIS
LIN {X 0.045,Y -175.533,Z 1773.411,A 0.000,B 0.000,C 90.000,E1 253.921} C_DIS
LIN {X 0.047,Y -172.268,Z 1773.387,A 0.000,B 0.000,C 90.000,E1 249.645} C_DIS
LIN {X 0.086,Y -171.747,Z 1773.382,A 0.000,B 0.000,C 90.000,E1 248.773} C_DIS
LIN {X -0.057,Y -167.345,Z 1773.353,A 0.000,B 0.000,C 90.000,E1 243.640} C_DIS
LIN {X 0.025,Y -166.732,Z 1773.349,A 0.000,B 0.000,C 90.000,E1 242.743} C_DIS
LIN {X -0.062,Y -162.711,Z 1773.324,A 0.000,B 0.000,C 90.000,E1 238.408} C_DIS
LIN {X -0.001,Y -161.402,Z 1773.315,A 0.000,B 0.000,C 90.000,E1 236.628} C_DIS
LIN {X 0.041,Y -157.395,Z 1773.290,A 0.000,B 0.000,C 90.000,E1 232.190} C_DIS
LIN {X -0.026,Y -155.392,Z 1773.275,A 0.000,B 0.000,C 90.000,E1 229.542} C_DIS
LIN {X 0.014,Y -151.726,Z 1773.250,A 0.000,B 0.000,C 90.000,E1 225.040} C_DIS
LIN {X 0.029,Y -149.920,Z 1773.235,A 0.000,B 0.000,C 90.000,E1 222.324} C_DIS
LIN {X -0.052,Y -146.774,Z 1773.210,A 0.000,B 0.000,C 90.000,E1 217.810} C_DIS
LIN {X 0.051,Y -145.344,Z 1773.195,A 0.000,B 0.000,C 90.000,E1 215.025} C_DIS
LIN {X -0.034,Y -142.420,Z 1773.164,A 0.000,B 0.000,C 90.000,E1 209.539} C_DIS
LIN {X 0.016,Y -141.405,Z 1773.149,A 0.000,B 0.000,C 90.000,E1 206.744} C_DIS
LIN {X 0.003,Y -139.356,Z 1773.113,A 0.000,B 0.000,C 90.000,E1 200.248} C_DIS
LIN {X -0.009,Y -138.799,Z 1773.097,A 0.000,B 0.000,C 90.000,E1 197.457} C_DIS
LIN {X 0.045,Y -138.348,Z 1773.055,A 0.000,B 0.000,C 90.000,E1 189.962} C_DIS
LIN {X 0.063,Y -139.370,Z 1773.009,A 0.000,B 0.000,C 90.000,E1 181.547} C_DIS
LIN {X -0.023,Y -141.260,Z 1772.973,A 0.000,B 0.000,C 90.000,E1 175.065} C_DIS
LIN {X -0.065,Y -142.627,Z 1772.957,A 0.000,B 0.000,C 90.000,E1 172.299} C_DIS
LIN {X 0.028,Y -144.950,Z 1772.931,A 0.000,B 0.000,C 90.000,E1 167.645} C_DIS
LIN {X 0.020,Y -147.579,Z 1772.911,A 0.000,B 0.000,C 90.000,E1 163.976} C_DIS
LIN {X 0.049,Y -150.190,Z 1772.891,A 0.000,B 0.000,C 90.000,E1 160.315} C_DIS
LIN {X -0.084,Y -153.571,Z 1772.871,A 0.000,B 0.000,C 90.000,E1 156.741} C_DIS
LIN {X -0.033,Y -156.987,Z 1772.851,A 0.000,B 0.000,C 90.000,E1 153.127} C_DIS
LIN {X 0.040,Y -161.101,Z 1772.831,A 0.000,B 0.000,C 90.000,E1 149.537} C_DIS
LIN {X -0.015,Y -163.205,Z 1772.821,A 0.000,B 0.000,C 90.000,E1 147.788} C_DIS
LIN {X -0.010,Y -167.632,Z 1772.802,A 0.000,B 0.000,C 90.000,E1 144.276} C_DIS
LIN {X 0.005,Y -171.458,Z 1772.787,A 0.000,B 0.000,C 90.000,E1 141.662} C_DIS
LIN {X -0.064,Y -176.382,Z 1772.768,A 0.000,B 0.000,C 90.000,E1 138.243} C_DIS
LIN {X 0.058,Y -180.676,Z 1772.754,A 0.000,B 0.000,C 90.000,E1 135.648} C_DIS
LIN {X 0.041,Y -186.078,Z 1772.735,A 0.000,B 0.000,C 90.000,E1 132.285} C_DIS
LIN {X -0.023,Y -190.715,Z 1772.721,A 0.000,B 0.000,C 90.000,E1 129.806} C_DIS
LIN {X 0.009,Y -196.468,Z 1772.703,A 0.000,B 0.000,C 90.000,E1 126.503} C_DIS
LIN {X -0.025,Y -201.249,Z 1772.689,A 0.000,B 0.000,C 90.000,E1 124.072} C_DIS
LIN {X 0.008,Y -207.208,Z 1772.671,A 0.000,B 0.000,C 90.000,E1 120.846} C_DIS
LIN {X 0.054,Y -210.887,Z 1772.661,A 0.000,B 0.000,C 90.000,E1 118.999} C_DIS
LIN {X 0.051,Y -337.566,Z 1772.661,A 0.000,B 0.000,C 90.000,E1 118.999} C_DIS
LIN {X 0.137,Y -339.573,Z 1772.661,A 0.000,B 0.000,C 90.000,E1 118.949} C_DIS
LIN {X 0.150,Y -344.725,Z 1772.660,A 0.000,B 0.000,C 90.000,E1 118.693} C_DIS
LIN {X -0.141,Y -347.535,Z 1772.658,A 0.000,B 0.000,C 90.000,E1 118.487} C_DIS
LIN {X -0.116,Y -351.189,Z 1772.655,A 0.000,B 0.000,C 90.000,E1 117.975} C_DIS
LIN {X 0.044,Y -367.575,Z 1772.637,A 0.000,B 0.000,C 90.000,E1 114.643} C_DIS
LIN {X -0.081,Y -382.598,Z 1772.622,A 0.000,B 0.000,C 90.000,E1 112.025} C_DIS
LIN {X 0.127,Y -397.369,Z 1772.610,A 0.000,B 0.000,C 90.000,E1 109.704} C_DIS
LIN {X 0.149,Y -417.550,Z 1772.594,A 0.000,B 0.000,C 90.000,E1 106.913} C_DIS
LIN {X -0.070,Y -434.429,Z 1772.582,A 0.000,B 0.000,C 90.000,E1 104.773} C_DIS
LIN {X 0.201,Y -449.553,Z 1772.572,A 0.000,B 0.000,C 90.000,E1 102.883} C_DIS
LIN {X -0.128,Y -462.587,Z 1772.563,A 0.000,B 0.000,C 90.000,E1 101.366} C_DIS
LIN {X -0.012,Y -473.259,Z 1772.556,A 0.000,B 0.000,C 90.000,E1 100.074} C_DIS
LIN {X -0.177,Y -481.404,Z 1772.550,A 0.000,B 0.000,C 90.000,E1 99.086} C_DIS
LIN {X -0.210,Y -487.030,Z 1772.546,A 0.000,B 0.000,C 90.000,E1 98.341} C_DIS
LIN {X 0.052,Y -490.365,Z 1772.543,A 0.000,B 0.000,C 90.000,E1 97.814} C_DIS
LIN {X -0.221,Y -493.098,Z 1772.541,A 0.000,B 0.000,C 90.000,E1 97.352} C_DIS
LIN {X 0.105,Y -494.080,Z 1772.539,A 0.000,B 0.000,C 90.000,E1 97.068} C_DIS
LIN {X -0.141,Y -494.587,Z 1772.537,A 0.000,B 0.000,C 90.000,E1 96.606} C_DIS
LIN {X 0.121,Y -494.566,Z 1772.528,A 0.000,B 0.000,C 90.000,E1 95.106} C_DIS
LIN {X -0.123,Y -493.875,Z 1772.526,A 0.000,B 0.000,C 90.000,E1 94.645} C_DIS
LIN {X 0.088,Y -492.402,Z 1772.523,A 0.000,B 0.000,C 90.000,E1 94.131} C_DIS
LIN {X -0.160,Y -490.564,Z 1772.520,A 0.000,B 0.000,C 90.000,E1 93.669} C_DIS
LIN {X -0.225,Y -486.197,Z 1772.515,A 0.000,B 0.000,C 90.000,E1 92.694} C_DIS
LIN {X -0.037,Y -479.887,Z 1772.508,A 0.000,B 0.000,C 90.000,E1 91.432} C_DIS
LIN {X 0.050,Y -473.144,Z 1772.501,A 0.000,B 0.000,C 90.000,E1 90.172} C_DIS
LIN {X 0.036,Y -466.038,Z 1772.494,A 0.000,B 0.000,C 90.000,E1 88.912} C_DIS
LIN {X 0.174,Y -457.090,Z 1772.485,A 0.000,B 0.000,C 90.000,E1 87.364} C_DIS
LIN {X 0.180,Y -447.835,Z 1772.477,A 0.000,B 0.000,C 90.000,E1 85.812} C_DIS
LIN {X 0.030,Y -438.237,Z 1772.468,A 0.000,B 0.000,C 90.000,E1 84.261} C_DIS
LIN {X 0.185,Y -428.521,Z 1772.459,A 0.000,B 0.000,C 90.000,E1 82.648} C_DIS
LIN {X -0.044,Y -417.066,Z 1772.449,A 0.000,B 0.000,C 90.000,E1 80.792} C_DIS
LIN {X 0.087,Y -403.992,Z 1772.437,A 0.000,B 0.000,C 90.000,E1 78.578} C_DIS
LIN {X 0.041,Y -389.629,Z 1772.423,A 0.000,B 0.000,C 90.000,E1 76.061} C_DIS
LIN {X 0.016,Y -372.991,Z 1772.405,A 0.000,B 0.000,C 90.000,E1 72.906} C_DIS
LIN {X 0.051,Y -361.427,Z 1772.392,A 0.000,B 0.000,C 90.000,E1 70.550} C_DIS
LIN {X 0.052,Y -350.095,Z 1772.379,A 0.000,B 0.000,C 90.000,E1 68.156} C_DIS
LIN {X 0.051,Y -337.742,Z 1772.363,A 0.000,B 0.000,C 90.000,E1 65.409} C_DIS
LIN {X -0.076,Y -328.427,Z 1772.351,A 0.000,B 0.000,C 90.000,E1 63.256} C_DIS
LIN {X -0.198,Y -320.432,Z 1772.341,A 0.000,B 0.000,C 90.000,E1 61.385} C_DIS
LIN {X 0.114,Y -312.061,Z 1772.330,A 0.000,B 0.000,C 90.000,E1 59.410} C_DIS
LIN {X 0.110,Y -304.791,Z 1772.321,A 0.000,B 0.000,C 90.000,E1 57.788} C_DIS
LIN {X 0.176,Y -295.818,Z 1772.310,A 0.000,B 0.000,C 90.000,E1 55.801} C_DIS
LIN {X -0.142,Y -282.608,Z 1772.293,A 0.000,B 0.000,C 90.000,E1 52.844} C_DIS
LIN {X 0.078,Y -270.095,Z 1772.276,A 0.000,B 0.000,C 90.000,E1 49.703} C_DIS
LIN {X -0.090,Y -257.015,Z 1772.257,A 0.000,B 0.000,C 90.000,E1 46.215} C_DIS
LIN {X 0.061,Y -245.606,Z 1772.239,A 0.000,B 0.000,C 90.000,E1 42.933} C_DIS
LIN {X -0.054,Y -236.010,Z 1772.222,A 0.000,B 0.000,C 90.000,E1 40.011} C_DIS
LIN {X -0.020,Y -226.891,Z 1772.205,A 0.000,B 0.000,C 90.000,E1 36.996} C_DIS
LIN {X 0.078,Y -218.406,Z 1772.188,A 0.000,B 0.000,C 90.000,E1 33.913} C_DIS
LIN {X 0.093,Y -210.399,Z 1772.171,A 0.000,B 0.000,C 90.000,E1 30.797} C_DIS
LIN {X 0.060,Y -203.109,Z 1772.154,A 0.000,B 0.000,C 90.000,E1 27.641} C_DIS
LIN {X -0.065,Y -196.617,Z 1772.136,A 0.000,B 0.000,C 90.000,E1 24.463} C_DIS
LIN {X 0.037,Y -190.847,Z 1772.118,A 0.000,B 0.000,C 90.000,E1 21.173} C_DIS
LIN {X 0.033,Y -185.982,Z 1772.099,A 0.000,B 0.000,C 90.000,E1 17.873} C_DIS
LIN {X 0.032,Y -182.064,Z 1772.081,A 0.000,B 0.000,C 90.000,E1 14.537} C_DIS
LIN {X 0.080,Y -178.334,Z 1772.057,A 0.000,B 0.000,C 90.000,E1 10.310} C_DIS
LIN {X 0.009,Y -175.564,Z 1772.034,A 0.000,B 0.000,C 90.000,E1 6.087} C_DIS
LIN {X -0.026,Y -173.363,Z 1771.993,A 0.000,B 0.000,C 90.000,E1 358.682} C_DIS
LIN {X -0.085,Y -173.372,Z 1771.954,A 0.000,B 0.000,C 90.000,E1 351.837} C_DIS
LIN {X -0.011,Y -175.381,Z 1771.912,A 0.000,B 0.000,C 90.000,E1 344.102} C_DIS
LIN {X 0.089,Y -178.264,Z 1771.883,A 0.000,B 0.000,C 90.000,E1 338.954} C_DIS
LIN {X 0.028,Y -182.084,Z 1771.855,A 0.000,B 0.000,C 90.000,E1 333.896} C_DIS
LIN {X -0.018,Y -186.205,Z 1771.832,A 0.000,B 0.000,C 90.000,E1 329.715} C_DIS
LIN {X 0.027,Y -190.303,Z 1771.813,A 0.000,B 0.000,C 90.000,E1 326.373} C_DIS
LIN {X 0.004,Y -195.253,Z 1771.795,A 0.000,B 0.000,C 90.000,E1 323.084} C_DIS
LIN {X -0.016,Y -199.646,Z 1771.781,A 0.000,B 0.000,C 90.000,E1 320.642} C_DIS
LIN {X -0.106,Y -204.746,Z 1771.768,A 0.000,B 0.000,C 90.000,E1 318.243} C_DIS
LIN {X 0.056,Y -211.622,Z 1771.752,A 0.000,B 0.000,C 90.000,E1 315.405} C_DIS
LIN {X -0.025,Y -217.190,Z 1771.741,A 0.000,B 0.000,C 90.000,E1 313.461} C_DIS
LIN {X -0.010,Y -223.616,Z 1771.731,A 0.000,B 0.000,C 90.000,E1 311.515} C_DIS
LIN {X 0.040,Y -229.480,Z 1771.722,A 0.000,B 0.000,C 90.000,E1 309.967} C_DIS
LIN {X -0.009,Y -236.053,Z 1771.714,A 0.000,B 0.000,C 90.000,E1 308.463} C_DIS
LIN {X 0.042,Y -245.318,Z 1771.703,A 0.000,B 0.000,C 90.000,E1 306.583} C_DIS
LIN {X 0.106,Y -255.548,Z 1771.693,A 0.000,B 0.000,C 90.000,E1 304.739} C_DIS
LIN {X -0.084,Y -273.562,Z 1771.677,A 0.000,B 0.000,C 90.000,E1 301.926} C_DIS
LIN {X -0.002,Y -293.228,Z 1771.662,A 0.000,B 0.000,C 90.000,E1 299.155} C_DIS
LIN {X 0.060,Y -311.297,Z 1771.649,A 0.000,B 0.000,C 90.000,E1 296.821} C_DIS
LIN {X 0.096,Y -324.523,Z 1771.640,A 0.000,B 0.000,C 90.000,E1 295.207} C_DIS
LIN {X 0.002,Y -337.737,Z 1771.631,A 0.000,B 0.000,C 90.000,E1 293.643} C_DIS
LIN {X 0.106,Y -348.040,Z 1771.625,A 0.000,B 0.000,C 90.000,E1 292.386} C_DIS
LIN {X 0.128,Y -360.460,Z 1771.616,A 0.000,B 0.000,C 90.000,E1 290.865} C_DIS
LIN {X -0.097,Y -365.256,Z 1771.613,A 0.000,B 0.000,C 90.000,E1 290.301} C_DIS
LIN {X 0.001,Y -371.844,Z 1771.608,A 0.000,B 0.000,C 90.000,E1 289.396} C_DIS
LIN {X 0.190,Y -375.837,Z 1771.604,A 0.000,B 0.000,C 90.000,E1 288.779} C_DIS
LIN {X -0.078,Y -381.035,Z 1771.600,A 0.000,B 0.000,C 90.000,E1 287.946} C_DIS
LIN {X 0.181,Y -385.243,Z 1771.595,A 0.000,B 0.000,C 90.000,E1 287.040} C_DIS
LIN {X -0.030,Y -387.539,Z 1771.592,A 0.000,B 0.000,C 90.000,E1 286.496} C_DIS
LIN {X 0.144,Y -389.435,Z 1771.589,A 0.000,B 0.000,C 90.000,E1 285.898} C_DIS
LIN {X -0.155,Y -391.040,Z 1771.585,A 0.000,B 0.000,C 90.000,E1 285.371} C_DIS
LIN {X 0.038,Y -392.288,Z 1771.582,A 0.000,B 0.000,C 90.000,E1 284.773} C_DIS
LIN {X 0.142,Y -393.129,Z 1771.579,A 0.000,B 0.000,C 90.000,E1 284.189} C_DIS
LIN {X -0.032,Y -393.666,Z 1771.576,A 0.000,B 0.000,C 90.000,E1 283.647} C_DIS
LIN {X 0.088,Y -393.797,Z 1771.573,A 0.000,B 0.000,C 90.000,E1 283.063} C_DIS
LIN {X -0.171,Y -393.607,Z 1771.569,A 0.000,B 0.000,C 90.000,E1 282.535} C_DIS
LIN {X -0.045,Y -393.036,Z 1771.566,A 0.000,B 0.000,C 90.000,E1 281.951} C_DIS
LIN {X 0.082,Y -392.047,Z 1771.563,A 0.000,B 0.000,C 90.000,E1 281.366} C_DIS
LIN {X -0.180,Y -390.764,Z 1771.560,A 0.000,B 0.000,C 90.000,E1 280.838} C_DIS
LIN {X -0.064,Y -389.007,Z 1771.557,A 0.000,B 0.000,C 90.000,E1 280.254} C_DIS
LIN {X 0.087,Y -385.648,Z 1771.552,A 0.000,B 0.000,C 90.000,E1 279.378} C_DIS
LIN {X 0.142,Y -381.538,Z 1771.547,A 0.000,B 0.000,C 90.000,E1 278.511} C_DIS
LIN {X 0.156,Y -376.866,Z 1771.543,A 0.000,B 0.000,C 90.000,E1 277.644} C_DIS
